	IS_iErrorSource = 0
	IS_iExternWarns_RF = 0
	IS_strErrorSource[] = "VW-User"
	RETURN TRUE
ENDIF
bOk = TRUE
;
; 1: Manuelle Messunganmeldung wurde verwendet
IF (iExternWarns B_AND IS_STATE_WARN_MANMEAS) == IS_STATE_WARN_MANMEAS THEN
	;bisher gibt es kein Flag
	bOk = FALSE
ENDIF
;
; 2: bei Ergebnissimulation
IF (iExternWarns B_AND IS_STATE_WARN_EVAL) == IS_STATE_WARN_EVAL THEN
	;bisher gibt es kein Flag
	bOk = FALSE
ENDIF
;
; 3: Toleranzverletzung
IF (iExternWarns B_AND IS_STATE_WARN_TOL) == IS_STATE_WARN_TOL THEN
	$FLAG[IS_FLAG_WARN_TOL] = TRUE
	bOk = FALSE
ENDIF
;
RETURN bOK
;
ENDFCT
;---------------------------------------------------------------------------------------------
;ENDFOLD
;
;FOLD Zentrale Funktion zur Fehlerbehandlung
;---------------------------------------------------------------------------------------------
DEF IS_ProcessErrors()
DECL CHAR strErrorSource[10]
DECL INT OFFSET
DECL STATE_T STATE
CHAR ch_tempString[300]
;
IF (IS_iExternErrors==0) AND (IS_iInternErrors==0) THEN
	RETURN
ENDIF
;
IF (IS_iExternErrors <> 0) THEN
	SWITCH IS_iErrorSource
	CASE 1
		strErrorSource[] = "RoVis"
		strErrorSource[6] = 0
	CASE 2
		strErrorSource[] = "Genesis"
		strErrorSource[8] = 0
	CASE 3
		strErrorSource[] = "IQRob"
		strErrorSource[6] = 0
	CASE 4
		strErrorSource[] = "ISRob"
		strErrorSource[6] = 0
	CASE 5
		strErrorSource[] = "Dynalog"
		strErrorSource[8] = 0
		SWITCH IS_iExternErrors
			CASE 1
				IS_MSG_ERR(IS_MSG_ERR_RTC_CALIB)
			CASE 2
				SWITCH IS_iServiceMode
				CASE IS_iTOOL_CHANGE
					IS_MSG_ERR(IS_MSG_ERR_RTC_CALC_TOOL)
				CASE IS_iROBOT_CHANGE
					IS_MSG_ERR(IS_MSG_ERR_RTC_CALC_BASE)
				CASE IS_iSENSOR_CHANGE_IMT
					IS_MSG_ERR(IS_MSG_ERR_SERV_SENSIMT)
				DEFAULT
					IS_MSG_ERR(IS_MSG_ERR_RTC)
				ENDSWITCH
			DEFAULT
				IS_MSG_ERR(IS_MSG_ERR_RTC)
			ENDSWITCH
		RETURN
	DEFAULT
		strErrorSource[] = "ISRA"
		strErrorSource[5] = 0
	ENDSWITCH
;
	OFFSET=0
	SWRITE(IS_strErrorSource[], STATE, OFFSET, "%s%d", strErrorSource[], IS_iExternErrors)
ENDIF
;
IF (IS_iInternErrors <> 0) THEN
	strErrorSource[] = "VW-User"
	strErrorSource[8]= 0
	OFFSET=0
	SWRITE(IS_strErrorSource[], STATE, OFFSET, "%s%d", strErrorSource[], IS_iInternErrors)
ENDIF
;
IF (IS_iInternErrors == IS_Err_ID_Tolerance) THEN
	OFFSET=0
	SWRITE(ch_tempString[], STATE, OFFSET, "Max = {X %.2f, Y %.2f, Z %.2f, A %.2f, B %.2f, C %.2f}", IS_CORR_ACCEPT_FRAME.X, IS_CORR_ACCEPT_FRAME.Y, IS_CORR_ACCEPT_FRAME.Z, IS_CORR_ACCEPT_FRAME.A, IS_CORR_ACCEPT_FRAME.B, IS_CORR_ACCEPT_FRAME.C)
	IS_MSG_ERR(IS_MSG_ERR_TOL_EXCEEDED)
	RETURN
ENDIF
;
SWITCH IS_iServiceMode
	CASE IS_iSENSOR_CHANGE
		IF (IS_iErrorSource==3) AND (IS_iExternErrors==16) THEN
			;IS_MSG_ERR(IS_MSG_ERR_SERV_SENS2)
			IS_MSG(IS_MSG_I_TRANS_AXES, IS_MSG_TYPE_NOTIFY) ;Achswinkel werden uebertragen
			IS_iFnctID = 0
		ELSE
		  ;IS_MSG_ERR(IS_MSG_ERR_SERV_SENS2)
		ENDIF
		RETURN
	CASE IS_iTOOL_CHANGE
		IF (IS_iErrorSource==3) AND (IS_iExternErrors==16) THEN
			;IS_MSG_ERR(IS_MSG_ERR_AXIS1A)
			IS_MSG(IS_MSG_I_TRANS_AXES, IS_MSG_TYPE_NOTIFY) ;Achswinkel werden uebertragen
			IS_iFnctID = 0
		ELSE
		  IS_MSG_ERR(IS_MSG_ERR_SERV_TOOL)
		ENDIF
		RETURN
	CASE IS_iROBOT_CHANGE
		IF (IS_iErrorSource==3) AND (IS_iExternErrors==16) THEN
			;IS_MSG_ERR(IS_MSG_ERR_AXIS1A)
			IS_MSG(IS_MSG_I_TRANS_AXES, IS_MSG_TYPE_NOTIFY) ;Achswinkel werden uebertragen
			IS_iFnctID = 0
		ELSE
		  IF (IS_iErrorSource==3) AND (IS_iExternErrors==32) THEN
		  	;IS_MSG_ERR(IS_MSG_ERR_AXIS1B)
				IS_MSG(IS_MSG_I_TRANS_BASE, IS_MSG_TYPE_NOTIFY) ;Basedaten werden uebertragen
				IS_iFnctID = 0
			ELSE
			  IF (IS_iErrorSource==3) AND (IS_iExternErrors==48) THEN
					;IS_MSG_ERR(IS_MSG_ERR_AXIS1B)
					;IS_MSG_ERR(IS_MSG_ERR_AXIS1A)
					IS_MSG(IS_MSG_I_TRANS_BASE, IS_MSG_TYPE_NOTIFY) ;Basedaten werden uebertragen)
					IS_MSG(IS_MSG_I_TRANS_AXES, IS_MSG_TYPE_NOTIFY) ;Achswinkel werden uebertragen
					IS_iFnctID = 0
			  ELSE
				  IS_MSG_ERR(IS_MSG_ERR_SERV_ROB)
				ENDIF
			ENDIF
		ENDIF
		RETURN
   CASE IS_iSENSOR_CHANGE_IMT
		IS_MSG_ERR(IS_MSG_ERR_SERV_SENSIMT)
		IS_iFnctID = 0
		RETURN
ENDSWITCH
;
SWITCH IS_iFnctID
;
;FOLD SNYC
CASE IS_FnctID_IMT_Sync1
	IF (IS_iExternErrors>0) THEN
		IS_MSG_ERR(IS_MSG_ERR_SYNC1A)
	ELSE
		IS_MSG_ERR(IS_MSG_ERR_SYNC1B)
	ENDIF
CASE IS_FnctID_IMT_Sync2
	IF (IS_iExternErrors>0) THEN
		IS_MSG_ERR(IS_MSG_ERR_SYNC2A)
	ELSE
		IS_MSG_ERR(IS_MSG_ERR_SYNC2B)
	ENDIF
;ENDFOLD (SYNC)
;
;FOLD SELECT
CASE IS_FnctID_IMT_SelectUp1
IF (IS_iExternErrors>0) THEN
	IF (IS_iErrorSource==3) AND ((IS_iExternErrors b_and 4)==4) THEN
		IS_MSG_ERR(IS_MSG_ERR_SELECT1A, IS_MODEL)
	ELSE
		IS_MSG_ERR(IS_MSG_ERR_SELECT1, IS_MODEL)
	ENDIF
ELSE
	SWITCH IS_iInternErrors
		CASE IS_Err_ID_Drain 																;Ablauffehler
			IS_MSG_ERR(IS_MSG_ERR_SELECT1B, IS_MODEL)
		CASE IS_Err_ID_Timeout 															;Timeout
			IS_MSG_ERR(IS_MSG_ERR_SELECT1C)
		DEFAULT
			IS_MSG_ERR(IS_MSG_ERR_SELECT1, IS_MODEL)
	ENDSWITCH
ENDIF
CASE IS_FnctID_IMT_SelectUp2
		SWITCH IS_iInternErrors
			CASE IS_Err_ID_Drain
				IS_MSG_ERR(IS_MSG_ERR_SELECT2A)
			CASE IS_Err_ID_ProgID
				IS_MSG_ERR(IS_MSG_ERR_SELECT2B, IS_PROGID)
			DEFAULT
				IS_MSG_ERR(IS_MSG_ERR_SELECT2)
		ENDSWITCH
CASE IS_FnctID_IMT_SelectUp3
		SWITCH IS_iInternErrors
			CASE IS_Err_ID_Timeout
				IS_MSG_ERR(IS_MSG_ERR_SELECT3A, IS_PROGID)
			DEFAULT
			 IS_MSG_ERR(IS_MSG_ERR_SELECT3, IS_PROGID)
		ENDSWITCH
;ENDFOLD (SELECT)
;
;FOLD IMT_RREPARE
CASE IS_FnctID_IMT_Prepare
	IF (IS_iExternErrors>0) THEN
		IF ((IS_iExternErrors b_and 8)==8) THEN
			IS_MSG_ERR(IS_MSG_ERR_IMT_PREPARE1A, IS_SUBTYP)
		ELSE
			IS_MSG_ERR(IS_MSG_ERR_IMT_PREPARE1, IS_SUBTYP)
		ENDIF
	ELSE
		SWITCH IS_iInternErrors
			CASE IS_Err_ID_Timeout
				IS_MSG_ERR(IS_MSG_ERR_IMT_PREPARE1B, IS_SUBTYP)
			DEFAULT
				IS_MSG_ERR(IS_MSG_ERR_IMT_PREPARE1, IS_SUBTYP)
		ENDSWITCH
	ENDIF
;ENDFOLD (IMT_RREPARE)
;
;FOLD IMT_APPLY
CASE IS_FnctID_IMT_Apply
	IS_MSG_ERR(IS_MSG_ERR_IMT_APPLY, IS_SUBTYP)
;ENDFOLD (IMT_APPLY)
;
;FOLD ACHSWINKEL SENDEN
CASE IS_FnctID_IMT_SendAxis1
	IF (IS_iExternErrors>0) THEN
		IF ((IS_iExternErrors b_and 8)==8) THEN
			IS_MSG_ERR(IS_MSG_ERR_IMT_PREPARE1, IS_SUBTYP)
			IS_iFnctID = 0
			RETURN
		ENDIF
		IF (IS_iErrorSource==3) AND (IS_iExternErrors==16) THEN
		  IF (($MODE_OP==#T2) OR ($MODE_OP==#T1)) THEN
        ;MsgNotify("Achswinkel werden uebertragen", "ISRA")
      ENDIF
		ELSE
		  IF (IS_iErrorSource==3) AND (IS_iExternErrors==32) THEN
        IF (($MODE_OP==#T2) OR ($MODE_OP==#T1)) THEN
           ;MsgNotify("Basedaten werden uebertragen", "ISRA")
        ENDIF
			ELSE
			 IF (IS_iErrorSource==3) AND (IS_iExternErrors==48) THEN
         IF (($MODE_OP==#T2) OR ($MODE_OP==#T1)) THEN
            ;MsgNotify("Basedaten und Achswinkel werden uebertragen", "ISRA")
         ENDIF
			 ELSE
					IS_MSG_ERR(IS_MSG_ERR_AXIS1)
				ENDIF
			ENDIF
		ENDIF
	ELSE
		SWITCH IS_iInternErrors
			CASE IS_Err_ID_Drain
				IS_MSG_ERR(IS_MSG_ERR_AXIS1C)
			CASE IS_Err_ID_Timeout
				IS_MSG_ERR(IS_MSG_ERR_AXIS1D)
			DEFAULT
				IS_MSG_ERR(IS_MSG_ERR_AXIS1)
		ENDSWITCH
	ENDIF
CASE IS_FnctID_IMT_SendAxis2
	IF (IS_iExternErrors>0) THEN
		IF (IS_iErrorSource==3) AND (IS_iExternErrors==32) THEN
			IS_MSG_ERR(IS_MSG_ERR_AXIS1B)
		ELSE
			IS_MSG_ERR(IS_MSG_ERR_AXIS2)
		ENDIF
	ELSE
		SWITCH IS_iInternErrors
			CASE IS_Err_ID_Drain
				IS_MSG_ERR(IS_MSG_ERR_AXIS2A)
			CASE IS_Err_ID_Timeout
				IS_MSG_ERR(IS_MSG_ERR_AXIS2B)
			DEFAULT
				IS_MSG_ERR(IS_MSG_ERR_AXIS2)
		ENDSWITCH
	ENDIF
CASE IS_FnctID_IMT_SendAxis3
	IF (IS_iExternErrors>0) THEN
		IS_MSG_ERR(IS_MSG_ERR_AXIS3)
	ELSE
		SWITCH IS_iInternErrors
			CASE IS_Err_ID_Drain
				IS_MSG_ERR(IS_MSG_ERR_AXIS3A)
			CASE IS_Err_ID_Timeout
				IS_MSG_ERR(IS_MSG_ERR_AXIS3B)
			DEFAULT
				IS_MSG_ERR(IS_MSG_ERR_AXIS3)
		ENDSWITCH
	ENDIF
CASE IS_FnctID_IMT_SendAxis4
	IF (IS_iExternErrors>0) THEN
		IS_MSG_ERR(IS_MSG_ERR_AXIS4)
	ELSE
		SWITCH IS_iInternErrors
			CASE IS_Err_ID_Drain
				IS_MSG_ERR(IS_MSG_ERR_AXIS4A)
			CASE IS_Err_ID_Timeout
				IS_MSG_ERR(IS_MSG_ERR_AXIS4B)
			DEFAULT
				IS_MSG_ERR(IS_MSG_ERR_AXIS4)
		ENDSWITCH
	ENDIF
;ENDFOLD (ACHSEN)
;
;FOLD BASE SENDEN
CASE IS_FnctID_IMT_SendBase1
	IF (IS_iExternErrors>0) THEN
		IS_MSG_ERR(IS_MSG_ERR_BASE1)
	ELSE
		SWITCH IS_iInternErrors
			CASE IS_Err_ID_Drain
				IS_MSG_ERR(IS_MSG_ERR_BASE1A)
			CASE IS_Err_ID_Timeout
				IS_MSG_ERR(IS_MSG_ERR_BASE2B)
			DEFAULT
				IS_MSG_ERR(IS_MSG_ERR_BASE1)
		ENDSWITCH
	ENDIF
CASE IS_FnctID_IMT_SendBase2
	IF (IS_iExternErrors>0) THEN
		IS_MSG_ERR(IS_MSG_ERR_BASE2)
	ELSE
		SWITCH IS_iInternErrors
			CASE IS_Err_ID_Drain
				IS_MSG_ERR(IS_MSG_ERR_BASE2A)
			CASE IS_Err_ID_Timeout
				IS_MSG_ERR(IS_MSG_ERR_BASE2B)
			DEFAULT
				IS_MSG_ERR(IS_MSG_ERR_BASE2)
		ENDSWITCH
	ENDIF
CASE IS_FnctID_IMT_SendBase3
	IF (IS_iExternErrors>0) THEN
		IS_MSG_ERR(IS_MSG_ERR_BASE3)
	ELSE
		SWITCH IS_iInternErrors
			CASE IS_Err_ID_Drain
				IS_MSG_ERR(IS_MSG_ERR_BASE3A)
			CASE IS_Err_ID_Timeout
				IS_MSG_ERR(IS_MSG_ERR_BASE3B)
			DEFAULT
				IS_MSG_ERR(IS_MSG_ERR_BASE3)
		ENDSWITCH
	ENDIF
;ENDFOLD (BASE SENDEN)
;
;FOLD POSE SENDEN
CASE IS_FnctID_IMT_SendPose1
	IF (IS_iExternErrors>0) THEN
		IS_MSG_ERR(IS_MSG_ERR_POSE1)
	ELSE
		SWITCH IS_iInternErrors
			CASE IS_Err_ID_Drain
				IS_MSG_ERR(IS_MSG_ERR_POSE1A)
			CASE IS_Err_ID_Timeout
				IS_MSG_ERR(IS_MSG_ERR_POSE1B)
			DEFAULT
				IS_MSG_ERR(IS_MSG_ERR_POSE1)
		ENDSWITCH
	ENDIF
CASE IS_FnctID_IMT_SendPose2
	IF (IS_iExternErrors>0) THEN
		IS_MSG_ERR(IS_MSG_ERR_POSE2)
	ELSE
		SWITCH IS_iInternErrors
			CASE IS_Err_ID_Drain
				IS_MSG_ERR(IS_MSG_ERR_POSE2A)
			CASE IS_Err_ID_Timeout
				IS_MSG_ERR(IS_MSG_ERR_POSE2B)
			DEFAULT
				IS_MSG_ERR(IS_MSG_ERR_POSE2)
		ENDSWITCH
	ENDIF
CASE IS_FnctID_IMT_SendPose3
	IF (IS_iExternErrors>0) THEN
		IS_MSG_ERR(IS_MSG_ERR_POSE3)
	ELSE
		SWITCH IS_iInternErrors
			CASE IS_Err_ID_Drain
				IS_MSG_ERR(IS_MSG_ERR_POSE3A)
			CASE IS_Err_ID_Timeout
				IS_MSG_ERR(IS_MSG_ERR_POSE3B)
			DEFAULT
				IS_MSG_ERR(IS_MSG_ERR_POSE3)
		ENDSWITCH
	ENDIF
;ENDFOLD (POSE SENDEN)
;
;FOLD TOOL SENDEN
CASE IS_FnctID_IMT_SendTool1
	IF (IS_iExternErrors>0) THEN
		IS_MSG_ERR(IS_MSG_ERR_TOOL1)
	ELSE
		SWITCH IS_iInternErrors
			CASE IS_Err_ID_Drain
				IS_MSG_ERR(IS_MSG_ERR_TOOL1A)
			CASE IS_Err_ID_Timeout
				IS_MSG_ERR(IS_MSG_ERR_TOOL1B)
			DEFAULT
				IS_MSG_ERR(IS_MSG_ERR_TOOL1)
		ENDSWITCH
	ENDIF
CASE IS_FnctID_IMT_SendTool2
	IF (IS_iExternErrors>0) THEN
		IS_MSG_ERR(IS_MSG_ERR_TOOL2)
	ELSE
		SWITCH IS_iInternErrors
			CASE IS_Err_ID_Drain
				IS_MSG_ERR(IS_MSG_ERR_TOOL2A)
			CASE IS_Err_ID_Timeout
				IS_MSG_ERR(IS_MSG_ERR_TOOL2B)
			DEFAULT
				IS_MSG_ERR(IS_MSG_ERR_TOOL2)
		ENDSWITCH
	ENDIF
CASE IS_FnctID_IMT_SendTool3
	IF (IS_iExternErrors>0) THEN
		IS_MSG_ERR(IS_MSG_ERR_TOOL3)
	ELSE
		SWITCH IS_iInternErrors
			CASE IS_Err_ID_Drain
				IS_MSG_ERR(IS_MSG_ERR_TOOL3A)
			CASE IS_Err_ID_Timeout
				IS_MSG_ERR(IS_MSG_ERR_TOOL3B)
			DEFAULT
				IS_MSG_ERR(IS_MSG_ERR_TOOL3)
		ENDSWITCH
	ENDIF
;ENDFOLD (POSE SENDEN)
;
;FOLD END_POSE
CASE IS_FnctID_IMT_EndPose1, IS_FnctID_IMT_EndPose2
	IF (IS_iExternErrors>0) THEN
		IF ((IS_iExternErrors B_AND 64)==64) THEN
			IS_MSG_ERR(IS_MSG_ERR_IMT_END1A)
		ENDIF
		IF ((IS_iExternErrors B_AND 128)==128) THEN
			IS_MSG_ERR(IS_MSG_ERR_IMT_END1B)
		ELSE
			IS_MSG_ERR(IS_MSG_ERR_IMT_END1)
		ENDIF
	ELSE
		SWITCH IS_iInternErrors
			CASE IS_Err_ID_Timeout
				IS_MSG_ERR(IS_MSG_ERR_IMT_END1C)
			DEFAULT
				IS_MSG_ERR(IS_MSG_ERR_IMT_END1)
		ENDSWITCH
	ENDIF
;ENDFOLD (END_POSE)
;
;FOLD GetCorr
CASE IS_FnctID_IMT_GetCorr1
	IF (IS_iExternErrors>0) THEN
			IS_MSG_ERR(IS_MSG_ERR_GETCORR1)
	ELSE
		SWITCH IS_iInternErrors
			CASE IS_Err_ID_Drain
				IS_MSG_ERR(IS_MSG_ERR_GETCORR1A)
			CASE IS_Err_ID_Timeout
				IS_MSG_ERR(IS_MSG_ERR_GETCORR1B)
			DEFAULT
				IS_MSG_ERR(IS_MSG_ERR_GETCORR1)
		ENDSWITCH
	ENDIF
CASE IS_FnctID_IMT_GetCorr2
	IF (IS_iExternErrors>0) THEN
			IS_MSG_ERR(IS_MSG_ERR_GETCORR2)
	ELSE
		SWITCH IS_iInternErrors
			CASE IS_Err_ID_Drain
				IS_MSG_ERR(IS_MSG_ERR_GETCORR2A)
			CASE IS_Err_ID_Timeout
				IS_MSG_ERR(IS_MSG_ERR_GETCORR2B)
			DEFAULT
				IS_MSG_ERR(IS_MSG_ERR_GETCORR2)
		ENDSWITCH
	ENDIF
CASE IS_FnctID_IMT_GetCorr3
	IF (IS_iExternErrors>0) THEN
			IS_MSG_ERR(IS_MSG_ERR_GETCORR3)
	ELSE
		SWITCH IS_iInternErrors
			CASE IS_Err_ID_Drain
				IS_MSG_ERR(IS_MSG_ERR_GETCORR3A)
			CASE IS_Err_ID_Timeout
				IS_MSG_ERR(IS_MSG_ERR_GETCORR3B)
			DEFAULT
				IS_MSG_ERR(IS_MSG_ERR_GETCORR3)
		ENDSWITCH
	ENDIF
CASE IS_FnctID_IMT_GetCorr4
	IF (IS_iInternErrors == IS_Err_ID_Timeout) THEN
		IS_MSG_ERR(IS_MSG_ERR_GETCORR4A)
	ELSE
		IS_MSG_ERR(IS_MSG_ERR_GETCORR4)
	ENDIF
;ENDFOLD (GetCorr)
;
;FOLD RF_INIT
CASE IS_FnctID_RF_Init1
	IS_MSG_ERR(IS_MSG_ERR_RF_INIT1A)
CASE IS_FnctID_RF_Init2
	IS_MSG_ERR(IS_MSG_ERR_RF_INIT2A)
;ENDFOLD (RF_INIT)
;
;FOLD RF_Prepare
CASE IS_FnctID_RF_Prepare1
	IF (IS_iExternErrors>0) THEN
		IS_MSG_ERR(IS_MSG_ERR_RF_PREPARE1A, IS_TYP, IS_SUBTYP)
	ELSE
		IF (IS_iInternErrors == IS_Err_ID_Timeout) THEN
			IS_MSG_ERR(IS_MSG_ERR_RF_PREPARE1B, IS_TYP, IS_SUBTYP)
		ELSE
			IS_MSG_ERR(IS_MSG_ERR_RF_PREPARE1, IS_TYP, IS_SUBTYP)
		ENDIF
	ENDIF
CASE IS_FnctID_RF_Prepare2
	IF (IS_iExternErrors>0) THEN
		IS_MSG_ERR(IS_MSG_ERR_RF_PREPARE2A, IS_TYP, IS_SUBTYP)
	ELSE
		IF (IS_iInternErrors == IS_Err_ID_Timeout) THEN
			IS_MSG_ERR(IS_MSG_ERR_RF_PREPARE2B, IS_TYP, IS_SUBTYP)
		ELSE
			IS_MSG_ERR(IS_MSG_ERR_RF_PREPARE2, IS_TYP, IS_SUBTYP)
		ENDIF
	ENDIF
CASE IS_FnctID_RF_Prepare3
	IF (IS_iExternErrors>0) THEN
		IF ((IS_iExternErrors b_and IS_ErrBit_Prepare)==IS_ErrBit_Prepare) THEN
			IS_MSG_ERR(IS_MSG_ERR_RF_PREPARE3A, IS_TYP, IS_SUBTYP)
		ELSE
			IS_MSG_ERR(IS_MSG_ERR_RF_PREPARE3B, IS_TYP, IS_SUBTYP)
		ENDIF
	ELSE
		IF (IS_iInternErrors == IS_Err_ID_Timeout) THEN
			IS_MSG_ERR(IS_MSG_ERR_RF_PREPARE3C, IS_TYP, IS_SUBTYP)
		ELSE
			IS_MSG_ERR(IS_MSG_ERR_RF_PREPARE3, IS_TYP, IS_SUBTYP)
		ENDIF
	ENDIF
;ENDFOLD (RF_Prepare)
;
;FOLD RF_APPLY
CASE IS_FnctID_RF_Apply1
	IS_MSG_ERR(IS_MSG_ERR_RF_APPLY1, IS_TYP, IS_SUBTYP)
CASE IS_FnctID_RF_Apply2
	IF (IS_iExternErrors>0) THEN
			IS_MSG_ERR(IS_MSG_ERR_RF_APPLY2B, IS_TYP, IS_SUBTYP)
	ELSE
		IF (IS_iInternErrors == IS_Err_ID_Timeout) THEN
			IS_MSG_ERR(IS_MSG_ERR_RF_APPLY2A, IS_TYP, IS_SUBTYP)
		ELSE
			IS_MSG_ERR(IS_MSG_ERR_RF_APPLY2, IS_TYP, IS_SUBTYP)
		ENDIF
	ENDIF
CASE IS_FnctID_RF_Apply3
	IF (IS_iExternErrors>0) THEN
		IF ((IS_iExternErrors b_and IS_ErrBit_Feature)==IS_ErrBit_Feature) THEN
			IS_MSG_ERR(IS_MSG_ERR_RF_APPLY3C, IS_TYP, IS_SUBTYP)
			;IS_iFnctID = 0
			;RETURN
		ELSE
			IF ((IS_iExternErrors b_and IS_ErrBit_Tol)==IS_ErrBit_Tol) THEN
				IS_MSG_ERR(IS_MSG_ERR_RF_APPLY3D, IS_TYP, IS_SUBTYP)
				;IS_iFnctID = 0
				;RETURN
			ELSE
				IF ((IS_iExternErrors b_and IS_ErrBit_Deadly)==IS_ErrBit_Deadly) THEN
					IS_MSG_ERR(IS_MSG_ERR_RF_APPLY3E, IS_TYP, IS_SUBTYP)
					;IS_iFnctID = 0
					;RETURN
				ELSE
					IS_MSG_ERR(IS_MSG_ERR_RF_APPLY3B, IS_TYP, IS_SUBTYP)
				ENDIF
			ENDIF
		ENDIF
	ELSE
		IF (IS_iInternErrors == IS_Err_ID_Timeout) THEN
			IS_MSG_ERR(IS_MSG_ERR_RF_APPLY3A, IS_TYP, IS_SUBTYP)
		ELSE
			IS_MSG_ERR(IS_MSG_ERR_RF_APPLY3, IS_TYP, IS_SUBTYP)
		ENDIF
	ENDIF
CASE IS_FnctID_RF_Apply4
	IF (IS_iExternErrors>0) THEN
		IF ((IS_iExternErrors b_and IS_ErrBit_Feature)==IS_ErrBit_Feature) THEN
			IS_MSG_ERR(IS_MSG_ERR_RF_APPLY4C, IS_TYP, IS_SUBTYP)
			;IS_iFnctID = 0
			;RETURN
		ELSE
			IF ((IS_iExternErrors b_and IS_ErrBit_Tol)==IS_ErrBit_Tol) THEN
				IS_MSG_ERR(IS_MSG_ERR_RF_APPLY4D, IS_TYP, IS_SUBTYP)
				;IS_iFnctID = 0
				;RETURN
			ELSE
				IF ((IS_iExternErrors b_and IS_ErrBit_Deadly)==IS_ErrBit_Deadly) THEN
					IS_MSG_ERR(IS_MSG_ERR_RF_APPLY4E, IS_TYP, IS_SUBTYP)
					;IS_iFnctID = 0
					;RETURN
				ELSE
					IS_MSG_ERR(IS_MSG_ERR_RF_APPLY4B, IS_TYP, IS_SUBTYP)
				ENDIF
			ENDIF
		ENDIF
	ELSE
		IF (IS_iInternErrors == IS_Err_ID_Timeout) THEN
			IS_MSG_ERR(IS_MSG_ERR_RF_APPLY4A, IS_TYP, IS_SUBTYP)
		ELSE
			IS_MSG_ERR(IS_MSG_ERR_RF_APPLY4, IS_TYP, IS_SUBTYP)
		ENDIF
	ENDIF
CASE IS_FnctID_RF_Apply5
	IF (IS_iExternErrors>0) THEN
		IF ((IS_iExternErrors b_and IS_ErrBit_Feature)==IS_ErrBit_Feature) THEN
			IS_MSG_ERR(IS_MSG_ERR_RF_APPLY5C, IS_TYP, IS_SUBTYP)
			;IS_iFnctID = 0
			;RETURN
		ELSE
			IF ((IS_iExternErrors b_and IS_ErrBit_Tol)==IS_ErrBit_Tol) THEN
				IS_MSG_ERR(IS_MSG_ERR_RF_APPLY5D, IS_TYP, IS_SUBTYP)
				;IS_iFnctID = 0
				;RETURN
			ELSE
				IF ((IS_iExternErrors b_and IS_ErrBit_Deadly)==IS_ErrBit_Deadly) THEN
					IS_MSG_ERR(IS_MSG_ERR_RF_APPLY5E, IS_TYP, IS_SUBTYP)
					;IS_iFnctID = 0
					;RETURN
				ELSE
					IS_MSG_ERR(IS_MSG_ERR_RF_APPLY5B, IS_TYP, IS_SUBTYP)
				ENDIF
			ENDIF
		ENDIF
	ELSE
		IF (IS_iInternErrors == IS_Err_ID_Timeout) THEN
			IS_MSG_ERR(IS_MSG_ERR_RF_APPLY5A, IS_TYP, IS_SUBTYP)
		ELSE
			IS_MSG_ERR(IS_MSG_ERR_RF_APPLY5, IS_TYP, IS_SUBTYP)
		ENDIF
	ENDIF
CASE IS_FnctID_RF_Apply6
	IS_MSG_ERR(IS_MSG_ERR_RF_APPLY6)
;ENDFOLD (RF_APPLY)
;
;FOLD RF_ENDPOSE
CASE IS_FnctID_RF_End1
	IF (IS_iExternErrors>0) THEN
		IF ((IS_iExternErrors b_and IS_ErrBit_Feature)==IS_ErrBit_Feature) THEN
			IS_MSG_ERR(IS_MSG_ERR_RF_END1B)
			;IS_iFnctID = 0
			;RETURN
		ELSE
			IF ((IS_iExternErrors b_and IS_ErrBit_Tol)==IS_ErrBit_Tol) THEN
				IS_MSG_ERR(IS_MSG_ERR_RF_END1C)
				;IS_iFnctID = 0
				;RETURN
			ELSE
				IF ((IS_iExternErrors b_and IS_ErrBit_Deadly)==IS_ErrBit_Deadly) THEN
					IS_MSG_ERR(IS_MSG_ERR_RF_END1E)
					;IS_iFnctID = 0
					;RETURN
				ELSE
					IS_MSG_ERR(IS_MSG_ERR_RF_END1A)
				ENDIF
			ENDIF
		ENDIF
	ELSE
		IF (IS_iInternErrors == IS_Err_ID_Timeout) THEN
			IS_MSG_ERR(IS_MSG_ERR_RF_END1D)
		ELSE
			IS_MSG_ERR(IS_MSG_ERR_RF_END1)
		ENDIF
	ENDIF
CASE IS_FnctID_RF_End2
	IF (IS_iExternErrors>0) THEN
		IF ((IS_iExternErrors b_and IS_ErrBit_Feature)==IS_ErrBit_Feature) THEN
			IS_MSG_ERR(IS_MSG_ERR_RF_END2B)
			;IS_iFnctID = 0
			;RETURN
		ELSE
			IF ((IS_iExternErrors b_and IS_ErrBit_Tol)==IS_ErrBit_Tol) THEN
				IS_MSG_ERR(IS_MSG_ERR_RF_END2C)
				;IS_iFnctID = 0
				;RETURN
			ELSE
				IF ((IS_iExternErrors b_and IS_ErrBit_Deadly)==IS_ErrBit_Deadly) THEN
					IS_MSG_ERR(IS_MSG_ERR_RF_END2E)
					;IS_iFnctID = 0
					;RETURN
				ELSE
					IS_MSG_ERR(IS_MSG_ERR_RF_END2A)
				ENDIF
			ENDIF
		ENDIF
	ELSE
		IF (IS_iInternErrors == IS_Err_ID_Timeout) THEN
			IS_MSG_ERR(IS_MSG_ERR_RF_END2D)
		ELSE
			IS_MSG_ERR(IS_MSG_ERR_RF_END2)
		ENDIF
	ENDIF
CASE IS_FnctID_RF_End2
	IS_MSG_ERR(IS_MSG_ERR_RF_END3)
;ENDFOLD (RF_ENDPOSE)
;
;FOLD RF_GETGORR
CASE IS_FnctID_RF_GCorr1
	IF (IS_iExternErrors>0) THEN
		IS_MSG_ERR(IS_MSG_ERR_RF_CORR1B)
	ELSE
		IF (IS_iInternErrors == IS_Err_ID_Timeout) THEN
			IS_MSG_ERR(IS_MSG_ERR_RF_CORR1A)
		ELSE
			IS_MSG_ERR(IS_MSG_ERR_RF_END1)
		ENDIF
	ENDIF
CASE IS_FnctID_RF_GCorr2
	IF (IS_iExternErrors>0) THEN
		IS_MSG_ERR(IS_MSG_ERR_RF_CORR2B)
	ELSE
		IF (IS_iInternErrors == IS_Err_ID_Timeout) THEN
			IS_MSG_ERR(IS_MSG_ERR_RF_CORR2A)
		ELSE
			IS_MSG_ERR(IS_MSG_ERR_RF_END2)
		ENDIF
	ENDIF
CASE IS_FnctID_RF_GCorr3
	IS_MSG_ERR(IS_MSG_ERR_RF_CORR3)
;ENDFOLD (RF_GETGORR)
;
;FOLD Service
CASE IS_FnctID_IMT_Service
	IF (IS_iInternErrors == IS_Err_ID_Timeout) THEN
		SWITCH IS_iServiceMode
			CASE IS_iSENSOR_CHANGE
				IS_MSG_ERR(IS_MSG_ERR_SERVICE1a)
			CASE IS_iTOOL_CHANGE
				IS_MSG_ERR(IS_MSG_ERR_SERVICE1b)
			CASE IS_iROBOT_CHANGE
				IS_MSG_ERR(IS_MSG_ERR_SERVICE1c)
			CASE IS_iSENSOR_CHANGE_IMT
				IS_MSG_ERR(IS_MSG_ERR_SERVICE1d)
		ENDSWITCH
	ELSE
		SWITCH IS_iServiceMode
			CASE IS_iSENSOR_CHANGE
				IS_MSG_ERR(IS_MSG_ERR_SERVICE1e)
			CASE IS_iTOOL_CHANGE
				IS_MSG_ERR(IS_MSG_ERR_SERVICE1f)
			CASE IS_iROBOT_CHANGE
				IS_MSG_ERR(IS_MSG_ERR_SERVICE1g)
			CASE IS_iSENSOR_CHANGE_IMT
				IS_MSG_ERR(IS_MSG_ERR_SERVICE1h)
		ENDSWITCH
	ENDIF
;ENDFOLD (Service)
;
;FOLD ProcessState
CASE IS_FnctID_IMT_GetExtStat
	IS_MSG_ERR(IS_MSG_ERR_IMT_APPLY, IS_SUBTYP)
;ENDFOLD (ProcessState)
;
ENDSWITCH
;
IS_iFnctID = 0
;
END
;---------------------------------------------------------------------------------------------
;ENDFOLD
;
;FOLD Ergebnis-Zustand abfragen
;---------------------------------------------------------------------------------------------
DEFFCT BOOL IS_IMT_GetExternState (iStateResult:OUT, iStateWarning:OUT)
DECL INT iStateResult
DECL INT iStateWarning
DECL BOOL b_RetVal
;
IS_iFnctID = IS_FnctID_IMT_GetExtStat
;
IS_TX8_DATA_ID 				= 58			;Zustandsabfrage
IS_TX1_DATA_REQUEST 	= TRUE
IS_TX1_HANDSHAKE 			= IS_ToggleHandshake()
;
IF (IS_Wait(#IS_ERROR_ID, TRUE, 0) == FALSE) THEN
	$FLAG[IS_FLAG_ERROR] = TRUE
	IS_SetInternError(IS_IntErr_StReq1)
	RETURN FALSE
ENDIF
;
IS_iErrorSource  	= IS_RX8_ERR_SYS_ID
IS_iExternErrors 	= IS_RX8_ERRORS
iStateResult  		= IS_RX8_STATE_RESULT
iStateWarning 		= IS_RX8_STATE_WARNING
;
IS_TX1_DATA_REQUEST 	= FALSE
IS_TX1_DATA_ACCEPTED 	= TRUE
IS_TX1_HANDSHAKE 			= IS_ToggleHandshake()
;
b_RetVal = IS_Wait(#IS_ERROR_ID, FALSE, 0)
;
IF (b_RetVal == FALSE) THEN
	$FLAG[IS_FLAG_ERROR] = TRUE
	IS_SetInternError(IS_IntErr_StReq2)
ENDIF
;
IS_TX8_DATA_ID 				= 0
IS_TX1_DATA_ACCEPTED 	= FALSE
;
RETURN b_RetVal
ENDFCT
;---------------------------------------------------------------------------------------------
;ENDFOLD
;
;FOLD Ergebniszustand auf Roboter Flags abbilden
;---------------------------------------------------------------------------------------------
DEFFCT BOOL IS_IMT_ProcessExtState (iExternStateResult:IN, iExternStateWarning:IN)
DECL INT iExternStateResult
DECL INT iExternStateWarning
;
IF (iExternStateResult B_AND IS_STATE_RESULT_OK) == IS_STATE_RESULT_OK THEN
	$FLAG[IS_FLAG_RESULT_OK]  = TRUE
	$FLAG[IS_FLAG_RESULT_NOK] = FALSE
ELSE
	$FLAG[IS_FLAG_RESULT_OK]	= FALSE
ENDIF
;
IF (iExternStateResult B_AND IS_STATE_RESULT_NOK) == IS_STATE_RESULT_NOK THEN
	$FLAG[IS_FLAG_RESULT_NOK] = TRUE
	$FLAG[IS_FLAG_RESULT_OK]  = FALSE
  IS_MSG_ERR(IS_MSG_RESULT_NOK)
  RETURN FALSE
ELSE
	$FLAG[IS_FLAG_RESULT_NOK]	= FALSE
  $FLAG[IS_FLAG_RESULT_OK]  = TRUE
ENDIF
;
IF (iExternStateWarning B_AND IS_STATE_WARN_TOL) == IS_STATE_WARN_TOL THEN
 	$FLAG[IS_FLAG_WARN_TOL] = TRUE
ELSE
  $FLAG[IS_FLAG_WARN_TOL] = FALSE
ENDIF
;
RETURN TRUE
ENDFCT
;---------------------------------------------------------------------------------------------
;ENDFOLD
;
;FOLD Systemdiagnose durchfuehren
;---------------------------------------------------------------------------------------------
DEF  IS_SYSTEM_DIAG ()
DECL BOOL bFlag
;
IF (IS_SYS_TYPE == IS_SYS_TYPE_IMT) THEN
	IF $IS_LIVE_SIGNAL THEN
		IS_MSG(IS_MSG_I_SYS_DIAG_1, IS_MSG_TYPE_NOTIFY)
	ELSE
		IS_MSG(IS_MSG_I_SYS_DIAG_2, IS_MSG_TYPE_NOTIFY)
		RETURN
	ENDIF
	;
	IF $IS_COMMUNICATE THEN
		IS_MSG(IS_MSG_I_SYS_DIAG_3, IS_MSG_TYPE_NOTIFY)
	ELSE
		IS_MSG(IS_MSG_I_SYS_DIAG_4, IS_MSG_TYPE_NOTIFY)
	ENDIF
	;
	;IS_MSG(0,7)
	IS_MSG(IS_MSG_I_SYNC, IS_MSG_TYPE_DIALOG)
	;
	IF (IS_ANSWER==1) THEN
		$IS_COMMUNICATE = TRUE
		IF IS_IMT_SyncHandshake() THEN
			IS_MSG(IS_MSG_I_SYS_DIAG_5, IS_MSG_TYPE_NOTIFY)
		ELSE
			IS_MSG(IS_MSG_I_SYS_DIAG_6, IS_MSG_TYPE_NOTIFY)
		ENDIF
	ELSE
		IS_MSG(IS_MSG_I_SYS_DIAG_7, IS_MSG_TYPE_NOTIFY)
	ENDIF
	;
ENDIF
;
IF (IS_SYS_TYPE == IS_SYS_TYPE_RF) THEN
	IF $IS_COMMUNICATE THEN
		IS_MSG(IS_MSG_I_SYS_DIAG_3, IS_MSG_TYPE_NOTIFY)
	ELSE
		IS_MSG(IS_MSG_I_SYS_DIAG_4, IS_MSG_TYPE_NOTIFY)
	ENDIF
	;
	;IS_MSG (0,7)
	IS_MSG(IS_MSG_I_SYNC, IS_MSG_TYPE_DIALOG)
	;
	IF (IS_ANSWER==1) THEN
		$IS_COMMUNICATE = TRUE
		;
		ISRA_PG_INIT()
		;
		IF IS_State_OK() THEN
			IS_MSG(IS_MSG_I_SYS_DIAG_5, IS_MSG_TYPE_NOTIFY)
		ELSE
			IS_MSG(IS_MSG_I_SYS_DIAG_6, IS_MSG_TYPE_NOTIFY)
		ENDIF
	ELSE
		IS_MSG(IS_MSG_I_SYS_DIAG_7, IS_MSG_TYPE_NOTIFY)
	ENDIF
ENDIF
;
END
;---------------------------------------------------------------------------------------------
;ENDFOLD
;
;
;FOLD HW über separate Messung prüfen
;---------------------------------------------------------------------------------------------
DEF IS_CheckHW()
	IF ((NOT IS_STATE_OK()) AND (NOT IS_bHWCheckMode) AND $IS_LIVE_SIGNAL) THEN
		;MsgNotify("IS_CheckHW", "Executing")
		; Fehlerflags speichern
		IS_SaveErrorFlags()
		;
		ISRA_PG_INIT()
		IS_bHWCheckMode = TRUE
		;
    IS_RF_Prepare(99, 0, 0)
    IS_RF_Apply(0)
    IS_RF_EndPose()
		;
		IF (NOT IS_STATE_OK()) AND (IS_RX1_RF_ERR_FEAT == TRUE) THEN
			$FLAG[IS_FLAG_ERR_ACQ] = TRUE
			$FLAG[IS_FLAG_ERROR] = TRUE
			IS_bHWCheckMode = FALSE
			IS_MSG_ERR(IS_MSG_ERR_RF_APPLY3E)
			;MsgNotify("IS_CheckHW","HW Error detected")
		ELSE
			IS_RestoreErrorFlags()
		ENDIF
	ENDIF
	IS_bHWCheckMode = FALSE
END
;---------------------------------------------------------------------------------------------
;ENDFOLD
;
;FOLD Speichern der Fehlerflags
;---------------------------------------------------------------------------------------------
DEF IS_SaveErrorFlags()
;
IS_FLAGS_SAVED[1] = $FLAG[IS_FLAG_ERR_SPS]
IS_FLAGS_SAVED[2] = $FLAG[IS_FLAG_ERR_ROBOT]
IS_FLAGS_SAVED[3] = $FLAG[IS_FLAG_ERR_PREPARE]
IS_FLAGS_SAVED[4] = $FLAG[IS_FLAG_ERR_ACQ]
IS_FLAGS_SAVED[5] = $FLAG[IS_FLAG_ERR_FEATURE]
IS_FLAGS_SAVED[6] = $FLAG[IS_FLAG_ERR_EVAL]
IS_FLAGS_SAVED[7] = $FLAG[IS_FLAG_ERR_TOL]
IS_FLAGS_SAVED[8] = $FLAG[IS_FLAG_WARN_TOL]
IS_FLAGS_SAVED[9] = $FLAG[IS_FLAG_KAL1_HLP]
IS_FLAGS_SAVED[10] = $FLAG[IS_FLAG_KAL2_HLP]
IS_FLAGS_SAVED[11] = $FLAG[IS_FLAG_RESULT_OK]
IS_FLAGS_SAVED[12] = $FLAG[IS_FLAG_RESULT_NOK]
IS_FLAGS_SAVED[13] = $FLAG[IS_FLAG_ERROR]
;
END
;---------------------------------------------------------------------------------------------
;ENDFOLD
;
;FOLD Wiederherstellen der Fehlerflags
;---------------------------------------------------------------------------------------------
DEF IS_RestoreErrorFlags()
;
$FLAG[IS_FLAG_ERR_SPS] 		= IS_FLAGS_SAVED[1]
$FLAG[IS_FLAG_ERR_ROBOT] 	= IS_FLAGS_SAVED[2]
$FLAG[IS_FLAG_ERR_PREPARE]= IS_FLAGS_SAVED[3]
$FLAG[IS_FLAG_ERR_ACQ]		= IS_FLAGS_SAVED[4]
$FLAG[IS_FLAG_ERR_FEATURE]= IS_FLAGS_SAVED[5]
$FLAG[IS_FLAG_ERR_EVAL]		= IS_FLAGS_SAVED[6]
$FLAG[IS_FLAG_ERR_TOL]		= IS_FLAGS_SAVED[7]
$FLAG[IS_FLAG_WARN_TOL]		= IS_FLAGS_SAVED[8]
$FLAG[IS_FLAG_KAL1_HLP]		= IS_FLAGS_SAVED[9]
$FLAG[IS_FLAG_KAL2_HLP]		= IS_FLAGS_SAVED[10]
$FLAG[IS_FLAG_RESULT_OK]	= IS_FLAGS_SAVED[11]
$FLAG[IS_FLAG_RESULT_NOK]	= IS_FLAGS_SAVED[12]
$FLAG[IS_FLAG_ERROR]			= IS_FLAGS_SAVED[13]
;
END
;---------------------------------------------------------------------------------------------
;ENDFOLD
;
;
;FOLD Fehlermeldungen deutsch
;---------------------------------------------------------------------------------------------
DEF  IS_MSG_ERR (iMsgNr:IN, iParam1:IN, iParam2:IN)
; Meldung die in allen Betriebsarten ausgegeben wird.
DECL INT iMsgNr
DECL INT MSG_QUIT_FLAG  ;Messages muessen quittiert werden.
DECL INT nHandle
DECL INT OFFSET
DECL STATE_T STATE
DECL CHAR MELDUNG[80]
DECL CHAR PARAM[10]
DECL INT IS_UserInstruction
CHAR ch_KXRKey[100]
CHAR ch_KXRKey_Btn1[10]
CHAR ch_KXRKey_Btn2[10]
DECL INT iParam1, iParam2
DECL KRLMSGPAR_T par1, par2

IS_UserInstruction=-1
;
IF IS_bHWCheckMode THEN
	RETURN
ENDIF
;
IF ($MODE_OP==#T1) OR ($MODE_OP==#T2) OR ((iMsgNr>=IS_IntErr_Param1) AND (iMsgNr<=IS_IntErr_Param6)) THEN
	MSG_QUIT_FLAG = 1
ELSE
	MSG_QUIT_FLAG = 2 ;Keine Quittierung in Automatik
ENDIF
;
;For Testing:
;MSG_QUIT_FLAG = 2
;
; Prepare the additional parameters
par1.par_type = #value
par2.par_type = #value
;
IF NOT (Varstate ("iParam1")==#initialized) then
   iParam1 = 0;
ENDIF
;
IF NOT (Varstate ("iParam2")==#initialized) then
   iParam2 = 0;
ENDIF
;
SWITCH iMsgNr
;Sync
CASE IS_MSG_ERR_SYNC1A
	ch_KXRKey[] = "IS_MSG_ERR_SYNC1A"
CASE IS_MSG_ERR_SYNC1B
	ch_KXRKey[] = "IS_MSG_ERR_SYNC1B"
	IS_UserInstruction = IS_Instr_Response
CASE IS_MSG_ERR_SYNC2A
	ch_KXRKey[] = "IS_MSG_ERR_SYNC2A"
CASE IS_MSG_ERR_SYNC2B
	ch_KXRKey[] = "IS_MSG_ERR_SYNC2B"
	IS_UserInstruction = IS_Instr_Response
;
;Select
CASE IS_MSG_ERR_SELECT1
	ch_KXRKey[] = "IS_MSG_ERR_SELECT1"
	IS_UserInstruction = IS_Instr_ModelCmp
CASE IS_MSG_ERR_SELECT1A
	ch_KXRKey[] = "IS_MSG_ERR_SELECT1A"
	IS_UserInstruction = IS_Instr_ModelChk
CASE IS_MSG_ERR_SELECT1B
	ch_KXRKey[] = "IS_MSG_ERR_SELECT1B"
	IS_UserInstruction = IS_Instr_DeadlyErr
CASE IS_MSG_ERR_SELECT1C
	ch_KXRKey[] = "IS_MSG_ERR_SELECT1C"
	IS_UserInstruction = IS_Instr_Response
CASE IS_MSG_ERR_SELECT2
	ch_KXRKey[] = "IS_MSG_ERR_SELECT2"
	IS_UserInstruction = IS_Instr_Response
CASE IS_MSG_ERR_SELECT2A
	ch_KXRKey[] = "IS_MSG_ERR_SELECT2A"
	IS_UserInstruction = IS_Instr_DeadlyErr
CASE IS_MSG_ERR_SELECT2B
	ch_KXRKey[] = "IS_MSG_ERR_SELECT2B"
CASE IS_MSG_ERR_SELECT3
	ch_KXRKey[] = "IS_MSG_ERR_SELECT3"
	IS_UserInstruction = IS_Instr_RoutCheck
CASE IS_MSG_ERR_SELECT3A
	ch_KXRKey[] = "IS_MSG_ERR_SELECT3A"
	IS_UserInstruction = IS_Instr_Response
;
;IMT Prepare
CASE IS_MSG_ERR_IMT_PREPARE1
	ch_KXRKey[] = "IS_MSG_ERR_IMT_PREPARE1"
CASE IS_MSG_ERR_IMT_PREPARE1A
	ch_KXRKey[] = "IS_MSG_ERR_IMT_PREPARE1A"
	IS_UserInstruction = IS_Instr_PntChk
CASE IS_MSG_ERR_IMT_PREPARE1B
	ch_KXRKey[] = "IS_MSG_ERR_IMT_PREPARE1B"
	IS_UserInstruction = IS_Instr_Response
;
;IMT_APPLY
CASE IS_MSG_ERR_IMT_APPLY
	ch_KXRKey[] = "IS_MSG_ERR_IMT_APPLY"
;
;Achsen senden
CASE IS_MSG_ERR_AXIS1
	ch_KXRKey[] = "IS_MSG_ERR_AXIS1"
CASE IS_MSG_ERR_AXIS1A
	ch_KXRKey[] = "IS_MSG_ERR_AXIS1A"
CASE IS_MSG_ERR_AXIS1B
	ch_KXRKey[] = "IS_MSG_ERR_AXIS1B"
CASE IS_MSG_ERR_AXIS1C
	ch_KXRKey[] = "IS_MSG_ERR_AXIS1C"
	IS_UserInstruction = IS_Instr_DeadlyErr
CASE IS_MSG_ERR_AXIS1D
	ch_KXRKey[] = "IS_MSG_ERR_AXIS1D"
	IS_UserInstruction = IS_Instr_Response
CASE IS_MSG_ERR_AXIS2
	ch_KXRKey[] = "IS_MSG_ERR_AXIS2"
	IS_UserInstruction = IS_Instr_DeadlyErr
CASE IS_MSG_ERR_AXIS2A
	ch_KXRKey[] = "IS_MSG_ERR_AXIS2A"
	IS_UserInstruction = IS_Instr_DeadlyErr
CASE IS_MSG_ERR_AXIS2B
	ch_KXRKey[] = "IS_MSG_ERR_AXIS2B"
	IS_UserInstruction = IS_Instr_Response
CASE IS_MSG_ERR_AXIS3
	ch_KXRKey[] = "IS_MSG_ERR_AXIS3"
	IS_UserInstruction = IS_Instr_DeadlyErr
CASE IS_MSG_ERR_AXIS3A
	ch_KXRKey[] = "IS_MSG_ERR_AXIS3A"
	IS_UserInstruction = IS_Instr_DeadlyErr
CASE IS_MSG_ERR_AXIS3B
	ch_KXRKey[] = "IS_MSG_ERR_AXIS3B"
	IS_UserInstruction = IS_Instr_Response
CASE IS_MSG_ERR_AXIS4
	ch_KXRKey[] = "IS_MSG_ERR_AXIS4"
	IS_UserInstruction = IS_Instr_DeadlyErr
CASE IS_MSG_ERR_AXIS4A
	ch_KXRKey[] = "IS_MSG_ERR_AXIS4A"
	IS_UserInstruction = IS_Instr_DeadlyErr
CASE IS_MSG_ERR_AXIS4B
	ch_KXRKey[] = "IS_MSG_ERR_AXIS4B"
	IS_UserInstruction = IS_Instr_Response
;
;Base senden
CASE IS_MSG_ERR_BASE1
	ch_KXRKey[] = "IS_MSG_ERR_BASE1"
	IS_UserInstruction = IS_Instr_DeadlyErr
CASE IS_MSG_ERR_BASE1A
	ch_KXRKey[] = "IS_MSG_ERR_BASE1A"
	IS_UserInstruction = IS_Instr_DeadlyErr
CASE IS_MSG_ERR_BASE1B
	ch_KXRKey[] = "IS_MSG_ERR_BASE2B"
	IS_UserInstruction = IS_Instr_Response
CASE IS_MSG_ERR_BASE2
	ch_KXRKey[] = "IS_MSG_ERR_BASE2"
	IS_UserInstruction = IS_Instr_DeadlyErr
CASE IS_MSG_ERR_BASE2A
	ch_KXRKey[] = "IS_MSG_ERR_BASE2A"
	IS_UserInstruction = IS_Instr_DeadlyErr
CASE IS_MSG_ERR_BASE2B
	ch_KXRKey[] = "IS_MSG_ERR_BASE2B"
	IS_UserInstruction = IS_Instr_Response
CASE IS_MSG_ERR_BASE3
	ch_KXRKey[] = "IS_MSG_ERR_BASE3"
	IS_UserInstruction = IS_Instr_DeadlyErr
CASE IS_MSG_ERR_BASE3A
	ch_KXRKey[] = "IS_MSG_ERR_BASE3A"
	IS_UserInstruction = IS_Instr_DeadlyErr
CASE IS_MSG_ERR_BASE3B
	ch_KXRKey[] = "IS_MSG_ERR_BASE3B"
	IS_UserInstruction = IS_Instr_Response
;
;IMT EndPose
CASE IS_MSG_ERR_IMT_END1
	ch_KXRKey[] = "IS_MSG_ERR_IMT_END1"
CASE IS_MSG_ERR_IMT_END1A
	ch_KXRKey[] = "IS_MSG_ERR_IMT_END1A"
CASE IS_MSG_ERR_IMT_END1B
	ch_KXRKey[] = "IS_MSG_ERR_IMT_END1B"
	IS_UserInstruction = IS_Instr_TolChk
CASE IS_MSG_ERR_IMT_END1C
	ch_KXRKey[] = "IS_MSG_ERR_IMT_END1C"
	IS_UserInstruction = IS_Instr_Response
;
;GetCorr
CASE IS_MSG_ERR_GETCORR1
	ch_KXRKey[] = "IS_MSG_ERR_GETCORR1"
	IS_UserInstruction = IS_Instr_DeadlyErr
CASE IS_MSG_ERR_GETCORR1A
	ch_KXRKey[] = "IS_MSG_ERR_GETCORR1A"
	IS_UserInstruction = IS_Instr_DeadlyErr
CASE IS_MSG_ERR_GETCORR1B
	ch_KXRKey[] = "IS_MSG_ERR_GETCORR1B"
	IS_UserInstruction = IS_Instr_Response
CASE IS_MSG_ERR_GETCORR2
	ch_KXRKey[] = "IS_MSG_ERR_GETCORR2"
	IS_UserInstruction = IS_Instr_DeadlyErr
CASE IS_MSG_ERR_GETCORR2A
	ch_KXRKey[] = "IS_MSG_ERR_GETCORR2A"
	IS_UserInstruction = IS_Instr_DeadlyErr
CASE IS_MSG_ERR_GETCORR2B
	ch_KXRKey[] = "IS_MSG_ERR_GETCORR2B"
	IS_UserInstruction = IS_Instr_Response
CASE IS_MSG_ERR_GETCORR3
	ch_KXRKey[] = "IS_MSG_ERR_GETCORR3"
	IS_UserInstruction = IS_Instr_DeadlyErr
CASE IS_MSG_ERR_GETCORR3A
	ch_KXRKey[] = "IS_MSG_ERR_GETCORR3A"
	IS_UserInstruction = IS_Instr_DeadlyErr
CASE IS_MSG_ERR_GETCORR3B
	ch_KXRKey[] = "IS_MSG_ERR_GETCORR3B"
	IS_UserInstruction = IS_Instr_Response
CASE IS_MSG_ERR_GETCORR4
	ch_KXRKey[] = "IS_MSG_ERR_GETCORR4"
	IS_UserInstruction = IS_Instr_DeadlyErr
CASE IS_MSG_ERR_GETCORR4A
	ch_KXRKey[] = "IS_MSG_ERR_GETCORR4A"
	IS_UserInstruction = IS_Instr_Response
;
CASE IS_MSG_ERR_TOL_EXCEEDED
	ch_KXRKey[] = "IS_MSG_ERR_TOL_EXCEEDED"
	IS_UserInstruction = IS_Instr_RobTol
;
;RF_Reset
CASE IS_MSG_ERR_RF_INIT1A
  ch_KXRKey[] = "IS_MSG_ERR_RF_INIT1A"
CASE IS_MSG_ERR_RF_INIT2A
  ch_KXRKey[] = "IS_MSG_ERR_RF_INIT2A"
;
;RF_Prepare
CASE IS_MSG_ERR_RF_PREPARE1
	ch_KXRKey[] = "IS_MSG_ERR_RF_PREPARE1"
	IS_UserInstruction = IS_Instr_DeadlyErr
CASE IS_MSG_ERR_RF_PREPARE1A
	ch_KXRKey[] = "IS_MSG_ERR_RF_PREPARE1A"
	IS_UserInstruction = IS_Instr_DeadlyErr
CASE IS_MSG_ERR_RF_PREPARE1B
	ch_KXRKey[] = "IS_MSG_ERR_RF_PREPARE1B"
	IS_UserInstruction = IS_Instr_Response
CASE IS_MSG_ERR_RF_PREPARE2
	ch_KXRKey[] = "IS_MSG_ERR_RF_PREPARE2"
	IS_UserInstruction = IS_Instr_DeadlyErr
CASE IS_MSG_ERR_RF_PREPARE2A
	ch_KXRKey[] = "IS_MSG_ERR_RF_PREPARE2A"
	IS_UserInstruction = IS_Instr_DeadlyErr
CASE IS_MSG_ERR_RF_PREPARE2B
	ch_KXRKey[] = "IS_MSG_ERR_RF_PREPARE2B"
	IS_UserInstruction = IS_Instr_Response
CASE IS_MSG_ERR_RF_PREPARE3
	ch_KXRKey[] = "IS_MSG_ERR_RF_PREPARE3"
	IS_UserInstruction = IS_Instr_DeadlyErr
CASE IS_MSG_ERR_RF_PREPARE3A
	ch_KXRKey[] = "IS_MSG_ERR_RF_PREPARE3A"
	IS_UserInstruction = IS_Instr_TypeChk
CASE IS_MSG_ERR_RF_PREPARE3B
	ch_KXRKey[] = "IS_MSG_ERR_RF_PREPARE3B"
	IS_UserInstruction = IS_Instr_DeadlyErr
CASE IS_MSG_ERR_RF_PREPARE3C
	ch_KXRKey[] = "IS_MSG_ERR_RF_PREPARE3C"
	IS_UserInstruction = IS_Instr_Response
;
;RF_APPLY
CASE IS_MSG_ERR_RF_APPLY1
	ch_KXRKey[] = "IS_MSG_ERR_RF_APPLY1"
	IS_UserInstruction = IS_Instr_DeadlyErr
;
CASE IS_MSG_ERR_RF_APPLY2
	ch_KXRKey[] = "IS_MSG_ERR_RF_APPLY2"
	IS_UserInstruction = IS_Instr_DeadlyErr
CASE IS_MSG_ERR_RF_APPLY2A
	ch_KXRKey[] = "IS_MSG_ERR_RF_APPLY2A"
	IS_UserInstruction = IS_Instr_Response
CASE IS_MSG_ERR_RF_APPLY2B
	ch_KXRKey[] = "IS_MSG_ERR_RF_APPLY2B"
	IS_UserInstruction = IS_Instr_DeadlyErr
;
CASE IS_MSG_ERR_RF_APPLY3
	ch_KXRKey[] = "IS_MSG_ERR_RF_APPLY3"
	IS_UserInstruction = IS_Instr_DeadlyErr
CASE IS_MSG_ERR_RF_APPLY3A
	ch_KXRKey[] = "IS_MSG_ERR_RF_APPLY3A"
	IS_UserInstruction = IS_Instr_Response
CASE IS_MSG_ERR_RF_APPLY3B
	ch_KXRKey[] = "IS_MSG_ERR_RF_APPLY3B"
	IS_UserInstruction = IS_Instr_ImgMsgChk
CASE IS_MSG_ERR_RF_APPLY3C
	ch_KXRKey[] = "IS_MSG_ERR_RF_APPLY3C"
	IS_UserInstruction = IS_Instr_ImgMsgChk
CASE IS_MSG_ERR_RF_APPLY3D
	ch_KXRKey[] = "IS_MSG_ERR_RF_APPLY3D"
	IS_UserInstruction = IS_Instr_TolChk
CASE IS_MSG_ERR_RF_APPLY3E
	ch_KXRKey[] = "IS_MSG_ERR_RF_APPLY3E"
	IS_UserInstruction = IS_Instr_HWChk
;
CASE IS_MSG_ERR_RF_APPLY4
	ch_KXRKey[] = "IS_MSG_ERR_RF_APPLY4"
	IS_UserInstruction = IS_Instr_DeadlyErr
CASE IS_MSG_ERR_RF_APPLY4A
	ch_KXRKey[] = "IS_MSG_ERR_RF_APPLY4A"
	IS_UserInstruction = IS_Instr_Response
CASE IS_MSG_ERR_RF_APPLY4B
	ch_KXRKey[] = "IS_MSG_ERR_RF_APPLY4B"
	IS_UserInstruction = IS_Instr_DeadlyErr
CASE IS_MSG_ERR_RF_APPLY4C
	ch_KXRKey[] = "IS_MSG_ERR_RF_APPLY4C"
	IS_UserInstruction = IS_Instr_ImgMsgChk
CASE IS_MSG_ERR_RF_APPLY4D
	ch_KXRKey[] = "IS_MSG_ERR_RF_APPLY4D"
	IS_UserInstruction = IS_Instr_TolChk
CASE IS_MSG_ERR_RF_APPLY4E
	ch_KXRKey[] = "IS_MSG_ERR_RF_APPLY4E"
	IS_UserInstruction = IS_Instr_HWChk
;
CASE IS_MSG_ERR_RF_APPLY5
	ch_KXRKey[] = "IS_MSG_ERR_RF_APPLY5"
	IS_UserInstruction = IS_Instr_DeadlyErr
CASE IS_MSG_ERR_RF_APPLY5A
	ch_KXRKey[] = "IS_MSG_ERR_RF_APPLY5A"
	IS_UserInstruction = IS_Instr_Response
CASE IS_MSG_ERR_RF_APPLY5B
	ch_KXRKey[] = "IS_MSG_ERR_RF_APPLY5B"
	IS_UserInstruction = IS_Instr_ImgMsgChk
CASE IS_MSG_ERR_RF_APPLY5C
	ch_KXRKey[] = "IS_MSG_ERR_RF_APPLY5C"
	IS_UserInstruction = IS_Instr_ImgMsgChk
CASE IS_MSG_ERR_RF_APPLY5D
	ch_KXRKey[] = "IS_MSG_ERR_RF_APPLY5D"
	IS_UserInstruction = IS_Instr_TolChk
CASE IS_MSG_ERR_RF_APPLY5E
	ch_KXRKey[] = "IS_MSG_ERR_RF_APPLY5E"
	IS_UserInstruction = IS_Instr_HWChk
;
CASE IS_MSG_ERR_RF_APPLY6
	ch_KXRKey[] = "IS_MSG_ERR_RF_APPLY6"
	IS_UserInstruction = IS_Instr_DeadlyErr
;
;RF_ENDPOSE
CASE IS_MSG_ERR_RF_END1
	ch_KXRKey[] = "IS_MSG_ERR_RF_END1"
	IS_UserInstruction = IS_Instr_DeadlyErr
CASE IS_MSG_ERR_RF_END1A
	ch_KXRKey[] = "IS_MSG_ERR_RF_END1A"
	IS_UserInstruction = IS_Instr_MsgChk
CASE IS_MSG_ERR_RF_END1B
	ch_KXRKey[] = "IS_MSG_ERR_RF_END1B"
	IS_UserInstruction = IS_Instr_ImgMsgChk
CASE IS_MSG_ERR_RF_END1C
	ch_KXRKey[] = "IS_MSG_ERR_RF_END1C"
	IS_UserInstruction = IS_Instr_TolChk
CASE IS_MSG_ERR_RF_END1D
	ch_KXRKey[] = "IS_MSG_ERR_RF_END1D"
	IS_UserInstruction = IS_Instr_Response
CASE IS_MSG_ERR_RF_END1E
  ch_KXRKey[] = "IS_MSG_ERR_RF_END1E"
  IS_UserInstruction = IS_Instr_HWChk
;
CASE IS_MSG_ERR_RF_END2
	ch_KXRKey[] = "IS_MSG_ERR_RF_END2"
	IS_UserInstruction = IS_Instr_DeadlyErr
CASE IS_MSG_ERR_RF_END2A
	ch_KXRKey[] = "IS_MSG_ERR_RF_END2A"
	IS_UserInstruction = IS_Instr_MsgChk
CASE IS_MSG_ERR_RF_END2B
	ch_KXRKey[] = "IS_MSG_ERR_RF_END2B"
	IS_UserInstruction = IS_Instr_MsgChk
CASE IS_MSG_ERR_RF_END2C
	ch_KXRKey[] = "IS_MSG_ERR_RF_END2C"
	IS_UserInstruction = IS_Instr_TolChk
CASE IS_MSG_ERR_RF_END2D
	ch_KXRKey[] = "IS_MSG_ERR_RF_END2D"
	IS_UserInstruction = IS_Instr_Response
CASE IS_MSG_ERR_RF_END2E
  ch_KXRKey[] = "IS_MSG_ERR_RF_END2E"
  IS_UserInstruction = IS_Instr_HWChk
;
CASE IS_MSG_ERR_RF_END3
	ch_KXRKey[] = "IS_MSG_ERR_RF_END3"
	IS_UserInstruction = IS_Instr_RobProg
;
;RF_GETCORRECTION
CASE IS_MSG_ERR_RF_CORR1
  ch_KXRKey[] = "IS_MSG_ERR_RF_CORR1"
  IS_UserInstruction = IS_Instr_DeadlyErr
CASE IS_MSG_ERR_RF_CORR1A
  ch_KXRKey[] = "IS_MSG_ERR_RF_CORR1A"
  IS_UserInstruction = IS_Instr_Response
CASE IS_MSG_ERR_RF_CORR1B
  ch_KXRKey[] = "IS_MSG_ERR_RF_CORR1B"
CASE IS_MSG_ERR_RF_CORR2
  ch_KXRKey[] = "IS_MSG_ERR_RF_CORR2"
  IS_UserInstruction = IS_Instr_DeadlyErr
CASE IS_MSG_ERR_RF_CORR2A
  ch_KXRKey[] = "IS_MSG_ERR_RF_CORR2A"
  IS_UserInstruction = IS_Instr_Response
CASE IS_MSG_ERR_RF_CORR2B
  ch_KXRKey[] = "IS_MSG_ERR_RF_CORR2B"
CASE IS_MSG_ERR_RF_CORR3
  ch_KXRKey[] = "IS_MSG_ERR_RF_CORR3"
;
;Service
CASE IS_MSG_ERR_SERV_SENS1
	ch_KXRKey[] = "IS_MSG_ERR_SERV_SENS1"
	IS_UserInstruction = 0
	IS_Apply_Service(3) ;3
CASE IS_MSG_ERR_SERV_SENS2
	ch_KXRKey[] = "IS_MSG_ERR_SERV_SENS2"
	IS_UserInstruction = 0
CASE IS_MSG_ERR_SERV_TOOL
	ch_KXRKey[] = "IS_MSG_ERR_SERV_TOOL"
	IS_UserInstruction = 0
CASE IS_MSG_ERR_SERV_TOOL_T
	ch_KXRKey[] = "IS_MSG_ERR_SERV_TOOL_T"
	IS_UserInstruction = IS_Instr_TolChk
CASE IS_MSG_ERR_SERV_ROB
	ch_KXRKey[] = "IS_MSG_ERR_SERV_ROB"
	IS_UserInstruction = 0
CASE IS_MSG_ERR_SERV_ROB_T
	ch_KXRKey[] = "IS_MSG_ERR_SERV_ROB_T"
	IS_UserInstruction = IS_Instr_TolChk
CASE IS_MSG_ERR_SERV_SENSIMT
	ch_KXRKey[] = "IS_MSG_ERR_SERV_SENSIMT"
CASE IS_MSG_ERR_SERVICE1A
	ch_KXRKey[] = "IS_MSG_ERR_SERVICE1A"
	IS_UserInstruction = IS_Instr_Response
CASE IS_MSG_ERR_SERVICE1B
	ch_KXRKey[] = "IS_MSG_ERR_SERVICE1B"
	IS_UserInstruction = IS_Instr_Response
CASE IS_MSG_ERR_SERVICE1C
	ch_KXRKey[] = "IS_MSG_ERR_SERVICE1C"
	IS_UserInstruction = IS_Instr_Response
CASE IS_MSG_ERR_SERVICE1D
	ch_KXRKey[] = "IS_MSG_ERR_SERVICE1D"
	IS_UserInstruction = IS_Instr_Response
CASE IS_MSG_ERR_SERVICE1E
	ch_KXRKey[] = "IS_MSG_ERR_SERVICE1E"
CASE IS_MSG_ERR_SERVICE1F
	ch_KXRKey[] = "IS_MSG_ERR_SERVICE1F"
CASE IS_MSG_ERR_SERVICE1G
	ch_KXRKey[] = "IS_MSG_ERR_SERVICE1G"
CASE IS_MSG_ERR_SERVICE1H
	ch_KXRKey[] = "IS_MSG_ERR_SERVICE1H"
;
CASE IS_MSG_ERR_RTC
	ch_KXRKey[] = "IS_MSG_ERR_RTC"
	IS_UserInstruction = IS_Instr_CalChk
CASE IS_MSG_ERR_RTC_CALIB
	ch_KXRKey[] = "IS_MSG_ERR_RTC_CALIB"
CASE IS_MSG_ERR_RTC_CALC_TOOL
	ch_KXRKey[] = "IS_MSG_ERR_RTC_CALC_TOOL"
CASE IS_MSG_ERR_RTC_CALC_BASE
	ch_KXRKey[] = "IS_MSG_ERR_RTC_CALC_BASE"
CASE IS_MSG_ERR_REQUEST
	ch_KXRKey[] = "IS_MSG_ERR_REQUEST"
CASE IS_MSG_ERR_BASE
	ch_KXRKey[] = "IS_MSG_ERR_BASE"
CASE IS_MSG_ERR_BIT_TRNS
	ch_KXRKey[] = "IS_MSG_ERR_BIT_TRNS"
CASE IS_MSG_ERR_TRANSM
	ch_KXRKey[] = "IS_MSG_ERR_TRANSM"
CASE IS_MSG_PP_WARN
	ch_KXRKey[] = "IS_MSG_PP_WARN"
CASE IS_MSG_PP_MOVEMODE
	ch_KXRKey[] = "IS_MSG_PP_MOVEMODE"
CASE IS_MSG_PP_TOL
	ch_KXRKey[] = "IS_MSG_PP_TOL"
CASE IS_MSG_PP_INVERSE
	ch_KXRKey[] = "IS_MSG_PP_INVERSE"
CASE IS_MSG_PP_FORWARD
	ch_KXRKey[] = "IS_MSG_PP_FORWARD"
CASE IS_MSG_PP_TEST_POSA
	ch_KXRKey[] = "IS_MSG_PP_TEST_POSA"
CASE IS_MSG_PP_TEST_POSK
	ch_KXRKey[] = "IS_MSG_PP_TEST_POSK"
CASE IS_MSG_DEBUG
	ch_KXRKey[] = "IS_MSG_DEBUG"
;
;Zustand/Warnung
CASE IS_MSG_RESULT_OK
  ch_KXRKey[] = "IS_MSG_RESULT_OK"
CASE IS_MSG_RESULT_NOK
  ch_KXRKey[] = "IS_MSG_RESULT_NOK"
CASE IS_MSG_WARN_TOL
  ch_KXRKey[] = "IS_MSG_WARN_TOL"
;
; Fehler und Meldungen von intern
CASE IS_IntErr_Param1
  ch_KXRKey[] = "IS_IntErr_Param1"
CASE IS_IntErr_Param2
  ch_KXRKey[] = "IS_IntErr_Param2"
CASE IS_IntErr_Param3
  ch_KXRKey[] = "IS_IntErr_Param3"
CASE IS_IntErr_Param4
  ch_KXRKey[] = "IS_IntErr_Param4"
CASE IS_IntErr_Param5
  ch_KXRKey[] = "IS_IntErr_Param5"
CASE IS_IntErr_Param6
  ch_KXRKey[] = "IS_IntErr_Param6"
;
CASE IS_IntErr_Com
	ch_KXRKey[] = "IS_IntErr_Com"
CASE IS_IntErr_ERequest
 ch_KXRKey[] = "IS_IntErr_ERequest"
CASE IS_IntErr_Meas
  ch_KXRKey[] = "IS_IntErr_Meas"
CASE IS_IntErr_Retry
  ch_KXRKey[] = "IS_IntErr_Retry"
CASE IS_IntErr_Data
  ch_KXRKey[] = "IS_IntErr_Data"
CASE IS_IntErr_Base
  ch_KXRKey[] = "IS_IntErr_Base"
CASE IS_IntErr_Tool
  ch_KXRKey[] = "IS_IntErr_Tool"
CASE IS_IntErr_ESendBit
 ch_KXRKey[] = "IS_IntErr_ESendBit"
CASE IS_IntErr_Specif
  ch_KXRKey[] = "IS_IntErr_Specif"
CASE IS_IntErr_SrvcExp
 	ch_KXRKey[] = "IS_IntErr_SrvcExp"
CASE IS_IntErr_StReq1
  ch_KXRKey[] = "IS_IntErr_StReq1"
CASE IS_IntErr_StReq2
  ch_KXRKey[] = "IS_IntErr_StReq2"
CASE IS_IntErr_ESend
 	ch_KXRKey[] = "IS_IntErr_ESend"
CASE IS_IntErr_IQRWait
 	ch_KXRKey[] = "IS_IntErr_IQRWait"
 	MSG_QUIT_FLAG = 3
CASE IS_IntErr_PCWait
 	ch_KXRKey[] = "IS_IntErr_PCWait"
 	MSG_QUIT_FLAG = 3
CASE IS_IntErr_TolRob
 	ch_KXRKey[] = "IS_IntErr_TolRob"
CASE IS_IntErr_RFAState
  ch_KXRKey[] = "IS_IntErr_RFAState"
CASE IS_IntErr_MeasPosNo
  ch_KXRKey[] = "IS_IntErr_MeasPosNo"
CASE IS_IntErr_RFGCSt
	ch_KXRKey[] = "IS_IntErr_RFGCSt"
CASE IS_IntErr_RFEPSt
	ch_KXRKey[] = "IS_IntErr_RFEPSt"
;
DEFAULT
   ch_KXRKey[] = "IS_MSG_ERR_DEFAULT"
ENDSWITCH
;
;Set Parameters:
par1.par_int = iParam1
par2.par_int = iParam2
;
SWITCH MSG_QUIT_FLAG
CASE 1
	IF (iMsgNr == IS_IntErr_Com) THEN
		;Dauerschleife bis Verbindung wieder da ist und der Ablauf normal weiter geht oder Option zum simulieren:
		IS_RF_ReconnectLoop()
	ELSE
 		OFFSET = 0
 		;
 		;Liegt eine Handlungsanweisung vor?
 		IF (IS_UserInstruction <> -1) THEN
	 	  REPEAT
	 	  	; Solange wiederholen bis Dialog mit OK/Weiter bestätigt wird.
	 	  	IF (IS_iServiceMode == IS_iSERVICE_NONE) THEN
	 	  		; Wenn nicht in Serviceprogramm, dann Button Info&Weiter, da Frage nach Messwiederholung folgt
	 	  		ch_KXRKey_Btn1[]="INFO"
					ch_KXRKey_Btn2[]="FORWARD"
	 	  		IS_ShowDialog(IS_ANSWER,ch_KXRKey_Btn1[],ch_KXRKey_Btn2[]," "," "," "," "," ",ch_KXRKey[], "vw_isr_usr_r", TRUE, par1, par2)
	 	  	ELSE
	 	  		; Wenn in Serviceprogramm, dann Button Info&OK
	 	  		ch_KXRKey_Btn1[]="INFO"
					ch_KXRKey_Btn2[]="OK"
	 	  		IS_ShowDialog(IS_ANSWER,ch_KXRKey_Btn1[],ch_KXRKey_Btn2[]," "," "," "," "," ",ch_KXRKey[], "vw_isr_usr_r", TRUE, par1, par2)
	 	  	ENDIF
		 		IS_ANSWER = 8-IS_ANSWER
				IF (IS_ANSWER == 1) THEN
					;'Info': Handlungsanweisung anzeigen
					IS_GetUserInstruction(IS_UserInstruction)
				ELSE
					;'OK': Beenden ohne Handlungsanweisung
				ENDIF
			UNTIL (IS_ANSWER <> 1)
 		ELSE
 			; Dialog ohne Info-Button anzeigen
 			ch_KXRKey_Btn2[]="OK"
 			IS_ShowDialog(IS_ANSWER," ",ch_KXRKey_Btn2[]," "," "," "," "," ",ch_KXRKey[], "vw_isr_usr_r", TRUE, par1, par2)
 		ENDIF
	ENDIF
CASE 2
  IS_ShowMessage(nHandle, #notify, ch_KXRKey[], "vw_isr_usr_r", iMsgNr, TRUE, par1, par2)
ENDSWITCH
;
END ;of IS_MSG_ERR
;---------------------------------------------------------------------------------------------
;ENDFOLD
;
;FOLD Meldungsausgabe (Info, Quittierung und Dialog)
;---------------------------------------------------------------------------------------------
DEF  IS_MSG(iMsgNr: IN, iMsgType: IN, iParam: IN)
DECL INT iMsgNr, iMsgType, iParam
DECL KRLMSGPAR_T par1
DECL INT nHandle
CHAR ch_KXRKey[100]
CHAR ch_KXRKey_btn1[10]
CHAR ch_KXRKey_btn2[10]
;
; Prepare the additional parameter
par1.par_type = #value

IF NOT (Varstate ("iParam")==#initialized) then
   iParam = 0;
ENDIF
;
IF (($MODE_OP==#T2) OR ($MODE_OP==#T1) OR (IS_iServiceMode <> IS_iSERVICE_NONE)) THEN
	SWITCH iMsgNr
	CASE IS_MSG_I_SERV_SENS_CHK
 	  ch_KXRKey[] = "IS_Info_Serv_Sens_Chk"
 	CASE IS_MSG_I_SERV_SENS
 		ch_KXRKey[] = "IS_Info_Serv_Sens"
 	CASE IS_MSG_I_SERV_TOOL
		ch_KXRKey[] = "IS_Info_Serv_Tool"
 	CASE IS_MSG_I_SERV_TOOL_PATH1
 		ch_KXRKey[] = "IS_Info_Serv_Tool_Path"
 	CASE IS_MSG_I_SERV_ROB
 	  ch_KXRKey[] = "IS_Info_Serv_Rob"
 	CASE IS_MSG_I_SERV_ROB_PATH1
 	  ch_KXRKey[] = "IS_Info_Serv_Rob_Path"
 	CASE IS_MSG_I_SERV_SENSIMT
 		ch_KXRKey[] = "IS_Info_Serv_Sens_IMT"
 	CASE IS_MSG_I_TRANS_AXES
 		ch_KXRKey[] = "IS_Info_Transfer_Axes"
	CASE IS_MSG_I_TRANS_BASE
		ch_KXRKey[] = "IS_Info_Transfer_Base"
	CASE IS_MSG_I_SYS_DIAG_1
		ch_KXRKey[] = "IS_Info_Sys_Diag_1"
	CASE IS_MSG_I_SYS_DIAG_2
		ch_KXRKey[] = "IS_Info_Sys_Diag_2"
	CASE IS_MSG_I_SYS_DIAG_3
		ch_KXRKey[] = "IS_Info_Sys_Diag_3"
	CASE IS_MSG_I_SYS_DIAG_4
		ch_KXRKey[] = "IS_Info_Sys_Diag_4"
	CASE IS_MSG_I_SYS_DIAG_5
		ch_KXRKey[] = "IS_Info_Sys_Diag_5"
  CASE IS_MSG_I_SYS_DIAG_6
		ch_KXRKey[] = "IS_Info_Sys_Diag_6"
	CASE IS_MSG_I_SYS_DIAG_7
 		ch_KXRKey[] = "IS_Info_Sys_Diag_7"
	CASE IS_MSG_I_SYNC
	  IF (IS_SYS_TYPE == IS_SYS_TYPE_IMT) THEN
	  	ch_KXRKey[] = "IS_Info_Sync_IMT"
	  ENDIF
	  IF (IS_SYS_TYPE == IS_SYS_TYPE_RF) THEN
	  	ch_KXRKey[] = "IS_Info_Sync_RF"
	  ENDIF
		ch_KXRKey_btn1[]= "YES"
		ch_KXRKey_btn2[]= "NO"
	CASE IS_MSG_I_MEAS_FAILED
	  IF (IS_SYS_TYPE == IS_SYS_TYPE_RF) THEN
			ch_KXRKey[] = "IS_Info_Meas_Failed"
			ch_KXRKey_btn1[]= "REPEAT"
			ch_KXRKey_btn2[]= "CANCEL"
		ENDIF
	CASE IS_MSG_I_SERV_TOOL_PATH2
	  IF (IS_SYS_TYPE == IS_SYS_TYPE_RF) THEN
			ch_KXRKey_btn1[]= "OK"
			ch_KXRKey_btn2[]= " "
			ch_KXRKey[] = "IS_Info_Tool_Path_2"
	  ENDIF
	CASE IS_MSG_I_SERV_ROB_PATH2
	  IF (IS_SYS_TYPE == IS_SYS_TYPE_RF) THEN
			ch_KXRKey_btn1[]= "OK"
			ch_KXRKey_btn2[]= " "
			ch_KXRKey[] = "IS_Info_Tool_Path_2"
	  ENDIF
	ENDSWITCH
	;
	; Set parameter
	par1.par_int = iParam
	;
	SWITCH iMsgType
		CASE IS_MSG_TYPE_DIALOG
			IS_ShowDialog(IS_ANSWER,ch_KXRKey_btn1[],ch_KXRKey_btn2[]," "," "," "," "," ",ch_KXRKey[], "vw_isr_usr_r", TRUE, par1)
			IS_ANSWER = 8-IS_ANSWER
		CASE IS_MSG_TYPE_NOTIFY
			IS_ShowMessage(nHandle, #notify, ch_KXRKey[], "vw_isr_usr_r", iMsgNr, TRUE, par1)
		CASE IS_MSG_TYPE_QUIT
			IS_ShowMessage(nHandle, #quit, ch_KXRKey[], "vw_isr_usr_r", iMsgNr, TRUE, par1)
		CASE IS_MSG_TYPE_STATE
			IS_ShowMessage(nHandle, #state, ch_KXRKey[], "vw_isr_usr_r", iMsgNr, TRUE, par1)
		DEFAULT
			IS_ShowMessage(nHandle, #notify, ch_KXRKey[], "vw_isr_usr_r", iMsgNr, TRUE, par1)
	ENDSWITCH
ENDIF
;
END ;of IS_MSG
;---------------------------------------------------------------------------------------------
;ENDFOLD
;
;FOLD Framemessage
;---------------------------------------------------------------------------------------------
DEF IS_MSG_FRAME2 (TYPE:IN, NR:IN, INFRAME:IN)
DECL FRAME INFRAME
DECL INT TYPE, NR
DECL INT OFFSET
DECL STATE_T STATE
DECL INT nHandle
DECL CHAR NAME[20]
DECL CHAR MELDUNG[80]
DECL CHAR ch_KXRkey[100]
DECL CHAR ABS[20]
;
SWITCH TYPE
  CASE 1
    NAME[]="Baseoffset"
    ABS[]="Differenz Basedaten"
  CASE 2
    NAME[]="Tooloffset"
    ABS[]="Differenz Tooldaten"
  CASE 3	;
    NAME[]="Base"
    ABS[]="Alte Basedaten"
  CASE 4
    NAME[]="Base"
    ABS[]="Neue Basedaten"
  CASE 5
    NAME[]="Tool"
    ABS[]="Alte Tooldaten"
  CASE 6
    NAME[]="Tool"
    ABS[]="Neue Tooldaten"
  CASE 7
    NAME[]="Base"
    ABS[]="Korrekturdaten"
  CASE 8
    NAME[]="Tool"
    ABS[]="Korrekturdaten"
  CASE 9
    NAME[]="Grenzwert"
    ABS[]="Korrekturdaten"
ENDSWITCH
;
	OFFSET=0
	IF (NR>0) THEN
  	SWRITE(MELDUNG[],STATE,OFFSET,"%s%d: X:%.1f,Y:%.1f,Z:%.1f,A:%.3f,B:%.3f,C:%.3f",NAME[],NR,INFRAME.x,INFRAME.y,INFRAME.z,INFRAME.a,INFRAME.b,INFRAME.c)
  	;SWRITE(MELDUNG[],STATE,OFFSET,"X:%.1f,Y:%.1f,Z:%.1f,A:%.3f,B:%.3f,C:%.3f",INFRAME.x,INFRAME.y,INFRAME.z,INFRAME.a,INFRAME.b,INFRAME.c)
  ELSE
  	SWRITE(MELDUNG[],STATE,OFFSET,"%s: X:%.1f,Y:%.1f,Z:%.1f,A:%.3f,B:%.3f,C:%.3f",NAME[],INFRAME.x,INFRAME.y,INFRAME.z,INFRAME.a,INFRAME.b,INFRAME.c)
 	ENDIF
;
  ;MsgState(nHandle, MELDUNG[], ABS[])
  IS_ShowMessage(nHandle, #state, MELDUNG[], ABS[], 1, TRUE)
;
END ;of IS_MSG_FRAME2()
;---------------------------------------------------------------------------------------------
;ENDFOLD
;
;FOLD ShowDialog
DEF IS_ShowDialog(nAnswer:OUT, sDialogSK1[]:IN,sDialogSK2[]:IN,sDialogSK3[]:IN,sDialogSK4[]:IN,sDialogSK5[]:IN,sDialogSK6[]:IN,sDialogSK7[]:IN,sText[]:IN, sModul[]:IN, bLog:IN, Par1:IN,Par2:IN,Par3:IN)
;************************************************************
;Function: Executes a dialog
;************************************************************
DECL KrlMsg_T Msg
DECL KrlMsgDlgSK_T Msg_SOFTKEY[7]
DECL INT nHandle,nMsgSel,nApplNum,nMsgTNr,count, len, nAnswer, nMsgNr
DECL BOOL bLog,Clear
DECL KrlMsgPar_T Par1,Par2,Par3, MsgPar[3]
DECL EKrlMsgType MsgType
DECL KrlMsgOpt_T MsgOpt
DECL CHAR sModul[], sText[], sDialogSK1[], sDialogSK2[], sDialogSK3[], sDialogSK4[], sDialogSK5[], sDialogSK6[], sDialogSK7[]

;set Parameter (if existent (otherwise "empty"))
ERR_CLEAR($Err)
ON_ERROR_PROCEED
MsgPar[1]=Par1
IF ($Err.Number<>0)THEN
  MsgPar[1].par_type=#empty
ENDIF
ERR_CLEAR($Err)
ON_ERROR_PROCEED
MsgPar[2]=Par2
IF ($Err.Number<>0)THEN
  MsgPar[2].par_type=#empty
ENDIF
ERR_CLEAR($Err)
ON_ERROR_PROCEED
MsgPar[3]=Par3
IF ($Err.Number<>0)THEN
  MsgPar[3].par_type=#empty
ENDIF

;set Option
;Vorlaufstopp
MsgOpt.Vl_Stop=FALSE
;Clear message on program reset
MsgOpt.Clear_P_Reset=TRUE
;Clear message on block selection
MsgOpt.Clear_p_SAW=FALSE
;Log message
MsgOpt.Log_To_DB=bLog

;Standard aus MSGLIB
Msg.Nr=1
ERR_CLEAR($Err)
ON_ERROR_PROCEED
Msg.Nr=nMsgNr
len=Strlen(sText[])
IF len>0 THEN
  IF len>80 THEN
    len=80
  ENDIF
  FOR count=1 TO len
    Msg.Msg_txt[count]=sText[count]
  ENDFOR
ELSE
  Msg.Msg_txt[]="parameter sText[] is missing"
ENDIF

len=Strlen(sModul[])
IF len>0 THEN
  IF len>24 THEN
    len=24
  ENDIF
  FOR count=1 TO len
    Msg.Modul[count]=sModul[count]
  ENDFOR
ELSE
  Msg.Modul[]="Appl"
ENDIF

;Set softkey text (1)
ERR_CLEAR($Err)
ON_ERROR_PROCEED
len=Strlen(sDialogSK1[])
IF $Err.Number==0 THEN
  IF len > 0 THEN
    IF len>24 THEN
      len=24
    ENDIF
    Msg_SOFTKEY[7].Sk_Type = #KEY
    FOR count=1 TO len
      Msg_SOFTKEY[7].Sk_txt[count] = sDialogSK1[count]
    ENDFOR
  ENDIF
ELSE
  FOR count=1 TO 24
    Msg_SOFTKEY[7].Sk_txt[count] = " "
  ENDFOR
ENDIF

;Set softkey text (2)
ERR_CLEAR($Err)
ON_ERROR_PROCEED
len=Strlen(sDialogSK2[])
IF $Err.Number==0 THEN
  len=Strlen(sDialogSK2[])
  IF len > 0 THEN
    IF len>24 THEN
      len=24
    ENDIF
    Msg_SOFTKEY[6].Sk_Type = #KEY
    FOR count=1 TO len
      Msg_SOFTKEY[6].Sk_txt[count] = sDialogSK2[count]
    ENDFOR
  ENDIF
ELSE
  FOR count=1 TO 24
    Msg_SOFTKEY[6].Sk_txt[count] = " "
  ENDFOR
ENDIF

;Set softkey text (3)
ERR_CLEAR($Err)
ON_ERROR_PROCEED
len=Strlen(sDialogSK3[])
IF $Err.Number==0 THEN
  len=Strlen(sDialogSK3[])
  IF len > 0 THEN
    IF len>24 THEN
      len=24
    ENDIF
    Msg_SOFTKEY[5].Sk_Type = #KEY
    FOR count=1 TO len
      Msg_SOFTKEY[5].Sk_txt[count] = sDialogSK3[count]
    ENDFOR
  ENDIF
ELSE
  FOR count=1 TO 24
    Msg_SOFTKEY[5].Sk_txt[count] = " "
  ENDFOR
ENDIF

;Set softkey text (4)
ERR_CLEAR($Err)
ON_ERROR_PROCEED
len=Strlen(sDialogSK4[])
IF $Err.Number==0 THEN
  len=Strlen(sDialogSK4[])
  IF len > 0 THEN
    IF len>24 THEN
      len=24
    ENDIF
    Msg_SOFTKEY[4].Sk_Type = #KEY
    FOR count=1 TO len
      Msg_SOFTKEY[4].Sk_txt[count] = sDialogSK4[count]
    ENDFOR
  ENDIF
ELSE
  FOR count=1 TO 24
    Msg_SOFTKEY[4].Sk_txt[count] = " "
  ENDFOR
ENDIF

;Set softkey text (5)
ERR_CLEAR($Err)
ON_ERROR_PROCEED
len=Strlen(sDialogSK5[])
IF $Err.Number==0 THEN
  len=Strlen(sDialogSK5[])
  IF len > 0 THEN
    IF len>24 THEN
      len=24
    ENDIF
    Msg_SOFTKEY[3].Sk_Type = #KEY
    FOR count=1 TO len
      Msg_SOFTKEY[3].Sk_txt[count] = sDialogSK5[count]
    ENDFOR
  ENDIF
ELSE
  FOR count=1 TO 24
    Msg_SOFTKEY[3].Sk_txt[count] = " "
  ENDFOR
ENDIF

;Set softkey text (6)
ERR_CLEAR($Err)
ON_ERROR_PROCEED
len=Strlen(sDialogSK6[])
IF $Err.Number==0 THEN
  len=Strlen(sDialogSK6[])
  IF len > 0 THEN
    IF len>24 THEN
      len=24
    ENDIF
    Msg_SOFTKEY[2].Sk_Type = #KEY
    FOR count=1 TO len
      Msg_SOFTKEY[2].Sk_txt[count] = sDialogSK6[count]
    ENDFOR
  ENDIF
ELSE
  FOR count=1 TO 24
    Msg_SOFTKEY[2].Sk_txt[count] = " "
  ENDFOR
ENDIF

;Set softkey text (7)
ERR_CLEAR($Err)
ON_ERROR_PROCEED
len=Strlen(sDialogSK7[])
IF $Err.Number==0 THEN
  len=Strlen(sDialogSK7[])
  IF len > 0 THEN
    IF len>24 THEN
      len=24
    ENDIF
    Msg_SOFTKEY[1].Sk_Type = #KEY
    FOR count=1 TO len
      Msg_SOFTKEY[1].Sk_txt[count] = sDialogSK7[count]
    ENDFOR
  ENDIF
ELSE
  FOR count=1 TO 24
    Msg_SOFTKEY[1].Sk_txt[count] = " "
  ENDFOR
ENDIF

CONTINUE
nHandle=SET_KRLDLG(Msg, MsgPar[], Msg_SOFTKEY[], MsgOpt)

If (nHandle > 0) THEN
  REPEAT
  CONTINUE
  WAIT SEC 0.5
  UNTIL((NOT Exists_KrlDlg(nHandle, nAnswer)))
  Clear=Clear_KrlMsg(nHANDLE)
ENDIF
;
END
;
;
DEF IS_ShowMessage(nHandle:OUT, MsgType:IN, sText[]:IN, sModul[]:IN, nMsgNr:IN, bLog:IN, Par1:IN, Par2:IN, Par3:IN)
;************************************************************
;Function: Executes a Message Send of the notify message
;************************************************************
DECL CHAR sText[], sModul[]
DECL KrlMsg_T Msg
DECL EKrlMsgType MsgType
DECL KrlMsgPar_T Par1, Par2, Par3, MsgPar[3]
DECL KrlMsgOpt_T MsgOpt
DECL BOOL bLog
DECL INT count, len, nHandle, nMsgNr

;set Parameter (if existent (otherwise "empty"))
ERR_CLEAR($Err)
ON_ERROR_PROCEED
MsgPar[1]=Par1
if ($Err.Number<>0)Then
  MsgPar[1].par_type=#empty
endif
ERR_CLEAR($Err)
ON_ERROR_PROCEED
  MsgPar[2]=Par2
if ($Err.Number<>0)Then
MsgPar[2].par_type=#empty
endif
ERR_CLEAR($Err)
ON_ERROR_PROCEED
  MsgPar[3]=Par3
if ($Err.Number<>0)Then
  MsgPar[3].par_type=#empty
endif

;set Option
;Vorlaufstopp
MsgOpt.Vl_Stop=FALSE
;Clear message on program reset
MsgOpt.Clear_P_Reset=TRUE
;Clear message on block selection
MsgOpt.Clear_p_SAW=FALSE
;Log message
MsgOpt.Log_To_DB=bLog

;set MessagNumber
Msg.Nr=nMsgNr
;set Msgtext
len=Strlen(sText[])
if len>0 then
	if len>80 then
		len=80
	endif
	for count=1 to len
		Msg.Msg_txt[count]=sText[count]
	endfor
else
	Msg.Msg_txt[]="Message text is missing"
endif
;setMsg-Modul
len=Strlen(sModul[])
if len>0 then
	if len>24 then
		len=24
	endif
	for count=1 to len
		Msg.Modul[count]=sModul[count]
	endfor
else
	Msg.Modul[]="Module name missing"
endif

CONTINUE
nHandle=Set_KrlMsg (MsgType, Msg, MsgPar[], MsgOpt)

END
;
;ENDFOLD (ISRA)

--- vw_isr_usr_r.dat ---
&ACCESS  RV
&COMMENT KS26
&PARAM DISKPATH = VW_User/Applikation/LM_Vision/Isra
&PARAM TPUSER_VERSION = 8.3.0
&PARAM EDITMASK = vw_isr_usr_r
&REL 59
DEFDAT  vw_isr_usr_r PUBLIC
;
;***************************************************
;* ISRA                                            *
;* Version 1.30  / VKRC 4                          *
;* Bearbeitet am:                                  *
;* 27.11.2014 JHo                                  *
;***************************************************
;
;FOLD IN-Signals IMT
; ;BYTE 0-3 / 4-7
SIGNAL IS_RX32_CORR_X $IN[1953]  TO $IN[1984] ;DATA-ID 52
SIGNAL IS_RX32_CORR_Y $IN[1985]  TO $IN[2016] ;DATA-ID 52
SIGNAL IS_RX32_CORR_Z $IN[1953]  TO $IN[1984] ;DATA-ID 53
SIGNAL IS_RX32_CORR_A $IN[1985]  TO $IN[2016] ;DATA-ID 53
SIGNAL IS_RX32_CORR_B $IN[1953]  TO $IN[1984] ;DATA-ID 54
SIGNAL IS_RX32_CORR_C $IN[1985]  TO $IN[2016] ;DATA-ID 54
;
SIGNAL IS_RX32_TOOL_X $IN[1953]  TO $IN[1984] ;DATA-ID 55
SIGNAL IS_RX32_TOOL_Y $IN[1985]  TO $IN[2016] ;DATA-ID 55
SIGNAL IS_RX32_TOOL_Z $IN[1953]  TO $IN[1984] ;DATA-ID 56
SIGNAL IS_RX32_TOOL_A $IN[1985]  TO $IN[2016] ;DATA-ID 56
SIGNAL IS_RX32_TOOL_B $IN[1953]  TO $IN[1984] ;DATA-ID 57
SIGNAL IS_RX32_TOOL_C $IN[1985]  TO $IN[2016] ;DATA-ID 57
;
;Error
SIGNAL IS_RX8_ERR_SYS_ID $IN[1953]  TO $IN[1960] ;DATA-ID 9/58
SIGNAL IS_RX8_ERRORS $IN[1961]  TO $IN[1968] ;DATA-ID 9/58
;
;State/Warnings
SIGNAL IS_RX8_STATE_RESULT $IN[1969]  TO $IN[1976] ;DATA-ID 58
SIGNAL IS_RX8_STATE_WARNING $IN[1977]  TO $IN[1984] ;DATA-ID 58
;
;BYTE 8
SIGNAL IS_RX8_DATA_ID $IN[2017]  TO $IN[2024]
;
;BYTE 9
SIGNAL IS_RX8_PROG_ID $IN[2025]  TO $IN[2032] ;Data-ID 51
;
;BYTE 10
SIGNAL IS_RX1_INIT_SIGNALS $IN[2033]
SIGNAL IS_RX1_SKIP $IN[2034]
SIGNAL IS_RX1_CONTINUE $IN[2035]
SIGNAL IS_RX1_MEAS_END $IN[2036] ;RF Messung Ende
;
;BYTE 11
SIGNAL IS_RX1_DATA_UNCHANGED $IN[2041]
SIGNAL IS_RX1_DATA_REQUEST $IN[2042]
SIGNAL IS_RX1_DATA_VALID $IN[2043]
SIGNAL IS_RX1_DATA_ACCEPTED $IN[2044]
SIGNAL IS_RX1_DATA_END_TRANS $IN[2045]
SIGNAL IS_RX1_ERROR_STATE $IN[2046]
SIGNAL IS_RX1_LIVE_SIGNAL $IN[2047]
SIGNAL IS_RX1_HANDSHAKE $IN[2048]
;
;ENDFOLD
;
;FOLD OUT-Signals IMT
;
;BYTE 0-3 / 4-7
SIGNAL IS_TX32_AXIS_1 $OUT[1953]  TO $OUT[1984] ;DATA-ID 1
SIGNAL IS_TX32_AXIS_2 $OUT[1985]  TO $OUT[2016] ;DATA-ID 1
SIGNAL IS_TX32_AXIS_3 $OUT[1953]  TO $OUT[1984] ;DATA-ID 2
SIGNAL IS_TX32_AXIS_4 $OUT[1985]  TO $OUT[2016] ;DATA-ID 2
SIGNAL IS_TX32_AXIS_5 $OUT[1953]  TO $OUT[1984] ;DATA-ID 3
SIGNAL IS_TX32_AXIS_6 $OUT[1985]  TO $OUT[2016] ;DATA-ID 3
;
SIGNAL IS_TX32_BASE_X $OUT[1953]  TO $OUT[1984] ;DATA-ID 4
SIGNAL IS_TX32_BASE_Y $OUT[1985]  TO $OUT[2016] ;DATA-ID 4
SIGNAL IS_TX32_BASE_Z $OUT[1953]  TO $OUT[1984] ;DATA-ID 5
SIGNAL IS_TX32_BASE_A $OUT[1985]  TO $OUT[2016] ;DATA-ID 5
SIGNAL IS_TX32_BASE_B $OUT[1953]  TO $OUT[1984] ;DATA-ID 6
SIGNAL IS_TX32_BASE_C $OUT[1985]  TO $OUT[2016] ;DATA-ID 6
;
SIGNAL IS_TX3_IMT_STATUS $OUT[1953]  TO $OUT[1960] ;DATA-ID 7
SIGNAL IS_TX6_IMT_TURN $OUT[1961]  TO $OUT[1968] ;DATA-ID 7
;
SIGNAL IS_TX8_MODEL_ID $OUT[1953]  TO $OUT[1960] ;DATA-ID 8
SIGNAL IS_TX8_ERROR_ID1 $OUT[1953]  TO $OUT[1960] ;DATA-ID 9
SIGNAL IS_TX8_ERROR_ID2 $OUT[1961]  TO $OUT[1968] ;DATA-ID 9
SIGNAL IS_TX16_SERVICE_ID $OUT[1953]  TO $OUT[1968] ;DATA-ID 10
;
SIGNAL IS_TX32_POSE_X $OUT[1953]  TO $OUT[1984] ;DATA-ID 11
SIGNAL IS_TX32_POSE_Y $OUT[1985]  TO $OUT[2016] ;DATA-ID 11
SIGNAL IS_TX32_POSE_Z $OUT[1953]  TO $OUT[1984] ;DATA-ID 12
SIGNAL IS_TX32_POSE_A $OUT[1985]  TO $OUT[2016] ;DATA-ID 12
SIGNAL IS_TX32_POSE_B $OUT[1953]  TO $OUT[1984] ;DATA-ID 13
SIGNAL IS_TX32_POSE_C $OUT[1985]  TO $OUT[2016] ;DATA-ID 13
;
SIGNAL IS_TX32_TOOL_X $OUT[1953]  TO $OUT[1984] ;DATA-ID 14
SIGNAL IS_TX32_TOOL_Y $OUT[1985]  TO $OUT[2016] ;DATA-ID 14
SIGNAL IS_TX32_TOOL_Z $OUT[1953]  TO $OUT[1984] ;DATA-ID 15
SIGNAL IS_TX32_TOOL_A $OUT[1985]  TO $OUT[2016] ;DATA-ID 15
SIGNAL IS_TX32_TOOL_B $OUT[1953]  TO $OUT[1984] ;DATA-ID 16
SIGNAL IS_TX32_TOOL_C $OUT[1985]  TO $OUT[2016] ;DATA-ID 16
;
;BYTE 8
SIGNAL IS_TX8_DATA_ID $OUT[2017]  TO $OUT[2024]
;
;BYTE 9
SIGNAL IS_TX8_POSE_ID $OUT[2025]  TO $OUT[2032]
;
;BYTE 10
SIGNAL IS_TX1_INIT_SIGNALS $OUT[2033]
SIGNAL IS_TX1_SKIP $OUT[2034]
SIGNAL IS_TX1_APPROACH_POSE $OUT[2035]
SIGNAL IS_TX1_IN_POSE $OUT[2036]
SIGNAL IS_TX1_IN_ENDPOSE $OUT[2037]
SIGNAL IS_TX1_TIMEOUT $OUT[2038]
;
;BYTE 11
SIGNAL IS_TX1_DATA_UNCHANGED $OUT[2041]
SIGNAL IS_TX1_DATA_REQUEST $OUT[2042]
SIGNAL IS_TX1_DATA_VALID $OUT[2043]
SIGNAL IS_TX1_DATA_ACCEPTED $OUT[2044]
SIGNAL IS_TX1_DATA_END_TRANS $OUT[2045]
SIGNAL IS_TX1_ERROR_STATE $OUT[2046]
SIGNAL IS_TX1_LIVE_BIT $OUT[2047]
SIGNAL IS_TX1_HANDSHAKE $OUT[2048]
;
;ENDFOLD
;
;FOLD IN-Signals RF
;
SIGNAL IS_RX4_RF_RM $IN[1953]  TO $IN[1956]
SIGNAL IS_RX1_RF_PREP_OK $IN[1960]
SIGNAL IS_RX1_RF_IMG_ACQ $IN[1957]
SIGNAL IS_RX1_RF_MEAS_RUN $IN[1958]
SIGNAL IS_RX1_RF_RES_RUN $IN[1959]
SIGNAL IS_RX1_RF_READY $IN[1961]
SIGNAL IS_RX1_RF_LIVE $IN[1962]
;
;Errors:
SIGNAL IS_RX1_RF_ERR_DEADLY $IN[1969]
SIGNAL IS_RX1_RF_ERR_PREP $IN[1973]
SIGNAL IS_RX1_RF_ERR_FEAT $IN[1972]
SIGNAL IS_RX1_RF_ERR_TOL $IN[1976]
SIGNAL IS_RX8_RF_ERR_SUM $IN[1969]  TO $IN[1976]
;
;Warnings:
SIGNAL IS_RX1_RF_W_MAN $IN[1977]
SIGNAL IS_RX1_RF_W_TOL $IN[1978]
SIGNAL IS_RX1_RF_W_EVAL $IN[1979]
;
;Result Data:
SIGNAL IS_RX16_RF_RES_X $IN[1985]  TO $IN[2000]
SIGNAL IS_RX16_RF_RES_Y $IN[2001]  TO $IN[2016]
SIGNAL IS_RX16_RF_RES_Z $IN[2017]  TO $IN[2032]
SIGNAL IS_RX16_RF_RES_RX $IN[2033]  TO $IN[2048]
SIGNAL IS_RX16_RF_RES_RY $IN[2049]  TO $IN[2064]
SIGNAL IS_RX16_RF_RES_RZ $IN[2065]  TO $IN[2080]
;
;ENDFOLD
;
;FOLD OUT-Signals RF
;
SIGNAL IS_TX4_RF_RM $OUT[1953]  TO $OUT[1956]
SIGNAL IS_TX1_RF_TYP_STR $OUT[1960]
SIGNAL IS_TX1_RF_START $OUT[1957]
SIGNAL IS_TX1_RF_SRESET $OUT[1958]
SIGNAL IS_TX1_RF_ERESET $OUT[1959]
SIGNAL IS_TX8_RF_TYP $OUT[1961]  TO $OUT[1968]
SIGNAL IS_TX8_RF_SUB_TYP $OUT[1969]  TO $OUT[1976]
SIGNAL IS_TX8_RF_COLOR_ID $OUT[1977]  TO $OUT[1984]
SIGNAL IS_TX1_RF_LIVE $OUT[1985]
;
SIGNAL IS_TX16_TYPE_ID $OUT[1953]  TO $OUT[1968] ;DATA-ID 8	;RF
SIGNAL IS_TX16_SUBTYPE_ID $OUT[1969]  TO $OUT[1984] ;DATA-ID 8	;RF
SIGNAL IS_TX16_COLOR_ID $OUT[1985]  TO $OUT[2000] ;DATA-ID 8	;RF
;
;ENDFOLD
;
;FOLD Constants
;
ENUM ISWaitType IS_NONE,IS_VALID,IS_ACCEPTED,IS_CONTINUE,IS_REQUEST,IS_END,IS_ERROR_ID,IS_RF_READY,IS_RF_RM,IS_RF_PREP,IS_RF_IMGACQ,IS_RF_MESRUN,IS_RF_ERESET,IS_RF_RESRUN
;
DECL REAL IS_RF_rScaleXYZ=10.0
DECL REAL IS_RF_rScaleABC=1000.0
DECL REAL IS_IMT_rScaleXYZ=100000.0
DECL REAL IS_IMT_rScaleABC=1000000.0
DECL REAL IS_IMT_rScaleAxis=1000000.0
DECL REAL IS_rSettlingTime=0.25 ; 250ms
;
DECL INT IS_iWaitTimerID=11
;
DECL INT IS_IMT_iRobStopTimerID=8
DECL INT IS_IMT_iRobStopTime=0
;
FRAME IS_CORR_ACCEPT_FRAME={X 20.0,Y 20.0,Z 20.0,A 5.0,B 5.0,C 5.0}
;
FRAME IS_ITERATION_THRESHOLD={X 0.0200000107,Y 0.0200000107,Z 0.0200000107,A 0.100000001,B 0.100000001,C 0.100000001}
;
;ENDFOLD
;
;FOLD Runtime Variables
;
DECL INT IS_ANSWER=2
CHAR IS_MG=" "
INT IS_MSG_I_LVL=0 ; 0-2 Message Level, um so hoeher das level, desto mehr meldungen.
;
DECL INT IS_MODUS
DECL INT IS_TYP
DECL INT IS_SUBTYP
DECL INT IS_SPECIFIER
DECL INT IS_TOOLNR
DECL INT IS_WIEDERHOLUNG
DECL INT IS_MODEL
DECL INT IS_PROGID
;
DECL INT IS_RX16_DATA[6]
;
DECL CHAR IS_strFnctName[20]
DECL CHAR IS_strErrText[32]
DECL CHAR IS_strErrorSource[10]
DECL CHAR IS_chCurrentFeature[100]
;
DECL BOOL IS_bHandshake=TRUE
DECL BOOL IS_bSkipFlag=FALSE
DECL BOOL IS_bTimeoutFlag=FALSE
DECL BOOL IS_bInternError
DECL BOOL IS_bSendBase=FALSE
DECL BOOL IS_bRepeatUpSel=FALSE
DECL BOOL IS_bMeasurementOK=FALSE
DECL BOOL IS_bSendAxes=TRUE
; HW error detection:
DECL BOOL IS_bHWCheckMode=FALSE
DECL BOOL IS_FLAGS_SAVED[13]
;
DECL INT IS_iCurrentUserError
DECL INT IS_iCurrentModel=70
DECL INT IS_iCurrentSub=70
DECL INT $IS_iHandshakeCounter=1
DECL INT IS_iErrorSource
DECL INT IS_iExternErrors
DECL INT IS_iInternErrors
DECL INT IS_iFnctID
DECL INT IS_iExternWarns_RF ;Warnzustände von RoVis für RF
;
DECL INT IS_iMeasPoint
;
DECL INT IS_iRM_Calib=1
;
DECL INT IS_iQuitFlag
;
DECL INT IS_iMaxNumIterations=1
;
DECL REAL IS_rMeasurementDelay
;
;ENDFOLD
;
;FOLD IDs
;
;Flags
DECL INT IS_FLAG_RESULT_OK=495
DECL INT IS_FLAG_RESULT_NOK=496
DECL INT IS_FLAG_ERROR=497
DECL INT IS_FLAG_ERR_SPS=498
DECL INT IS_FLAG_ERR_ROBOT=499
DECL INT IS_FLAG_ERR_PREPARE=500
DECL INT IS_FLAG_ERR_ACQ=501
DECL INT IS_FLAG_ERR_FEATURE=502
DECL INT IS_FLAG_ERR_EVAL=503
DECL INT IS_FLAG_ERR_TOL=504
DECL INT IS_FLAG_WARN_TOL=505
DECL INT IS_FLAG_KAL1_HLP=506
DECL INT IS_FLAG_KAL2_HLP=507
;
;Msg Type ID
DECL INT IS_MSG_TYPE_NOTIFY=1
DECL INT IS_MSG_TYPE_DIALOG=2
DECL INT IS_MSG_TYPE_QUIT=3
DECL INT IS_MSG_TYPE_STATE=4
;
;Msg ID User Instruction
DECL INT IS_MSG_PREP_INSTR=4002
DECL INT IS_MSG_ACQ_INSTR=4003
DECL INT IS_MSG_FEAT_INSTR=4004
DECL INT IS_MSG_EVAL_INSTR=4005
DECL INT IS_MSG_TOL_INSTR=4006
;
;Msg ID Info
DECL INT IS_MSG_I_SERV_SENS_CHK=2003
DECL INT IS_MSG_I_SERV_SENS=2004
DECL INT IS_MSG_I_SERV_TOOL=2005
DECL INT IS_MSG_I_SERV_TOOL_PATH1=2006
DECL INT IS_MSG_I_SERV_ROB=2007
DECL INT IS_MSG_I_SERV_ROB_PATH1=2008
DECL INT IS_MSG_I_SERV_SENSIMT=2009
DECL INT IS_MSG_I_TRANS_AXES=2010
DECL INT IS_MSG_I_TRANS_BASE=2011
DECL INT IS_MSG_I_SYS_DIAG_1=3000
DECL INT IS_MSG_I_SYS_DIAG_2=3001
DECL INT IS_MSG_I_SYS_DIAG_3=3002
DECL INT IS_MSG_I_SYS_DIAG_4=3003
DECL INT IS_MSG_I_SYS_DIAG_5=3004
DECL INT IS_MSG_I_SYS_DIAG_6=3005
DECL INT IS_MSG_I_SYS_DIAG_7=3006
DECL INT IS_MSG_I_SYNC=4001 ; 7
DECL INT IS_MSG_I_MEAS_FAILED=4002 ; 8
DECL INT IS_MSG_I_SERV_TOOL_PATH2=4003 ; 12
DECL INT IS_MSG_I_SERV_ROB_PATH2=4004 ; 13
;
;Msg ID Error
DECL INT IS_MSG_ERR_SYNC1A=200
DECL INT IS_MSG_ERR_SYNC1B=201
DECL INT IS_MSG_ERR_SYNC2A=202
DECL INT IS_MSG_ERR_SYNC2B=203
DECL INT IS_MSG_ERR_SELECT1=204
DECL INT IS_MSG_ERR_SELECT1A=205
DECL INT IS_MSG_ERR_SELECT1B=206
DECL INT IS_MSG_ERR_SELECT1C=207
DECL INT IS_MSG_ERR_SELECT2=208
DECL INT IS_MSG_ERR_SELECT2A=209
DECL INT IS_MSG_ERR_SELECT2B=210
DECL INT IS_MSG_ERR_SELECT3=211
DECL INT IS_MSG_ERR_SELECT3A=212
DECL INT IS_MSG_ERR_IMT_PREPARE1=213
DECL INT IS_MSG_ERR_IMT_PREPARE1A=214
DECL INT IS_MSG_ERR_IMT_PREPARE1B=215
DECL INT IS_MSG_ERR_IMT_APPLY=216
DECL INT IS_MSG_ERR_AXIS1=217
DECL INT IS_MSG_ERR_AXIS1A=218
DECL INT IS_MSG_ERR_AXIS1B=219
DECL INT IS_MSG_ERR_AXIS1C=220
DECL INT IS_MSG_ERR_AXIS1D=221
DECL INT IS_MSG_ERR_AXIS2=222
DECL INT IS_MSG_ERR_AXIS2A=223
DECL INT IS_MSG_ERR_AXIS2B=224
DECL INT IS_MSG_ERR_AXIS3=225
DECL INT IS_MSG_ERR_AXIS3A=226
DECL INT IS_MSG_ERR_AXIS3B=227
DECL INT IS_MSG_ERR_AXIS4=228
DECL INT IS_MSG_ERR_AXIS4A=229
DECL INT IS_MSG_ERR_AXIS4B=230
DECL INT IS_MSG_ERR_BASE1=231
DECL INT IS_MSG_ERR_BASE1A=232
DECL INT IS_MSG_ERR_BASE1B=233
DECL INT IS_MSG_ERR_BASE2=234
DECL INT IS_MSG_ERR_BASE2A=235
DECL INT IS_MSG_ERR_BASE2B=236
DECL INT IS_MSG_ERR_BASE3=237
DECL INT IS_MSG_ERR_BASE3A=238
DECL INT IS_MSG_ERR_BASE3B=239
DECL INT IS_MSG_ERR_IMT_END1=240
DECL INT IS_MSG_ERR_IMT_END1A=241
DECL INT IS_MSG_ERR_IMT_END1B=242
DECL INT IS_MSG_ERR_IMT_END1C=243
DECL INT IS_MSG_ERR_GETCORR1=244
DECL INT IS_MSG_ERR_GETCORR1A=245
DECL INT IS_MSG_ERR_GETCORR1B=246
DECL INT IS_MSG_ERR_GETCORR2=247
DECL INT IS_MSG_ERR_GETCORR2A=248
DECL INT IS_MSG_ERR_GETCORR2B=249
DECL INT IS_MSG_ERR_GETCORR3=250
DECL INT IS_MSG_ERR_GETCORR3A=251
DECL INT IS_MSG_ERR_GETCORR3B=252
DECL INT IS_MSG_ERR_GETCORR4=253
DECL INT IS_MSG_ERR_GETCORR4A=254
DECL INT IS_MSG_ERR_POSE1=255
DECL INT IS_MSG_ERR_POSE1A=256
DECL INT IS_MSG_ERR_POSE1B=257
DECL INT IS_MSG_ERR_POSE2=258
DECL INT IS_MSG_ERR_POSE2A=259
DECL INT IS_MSG_ERR_POSE2B=260
DECL INT IS_MSG_ERR_POSE3=261
DECL INT IS_MSG_ERR_POSE3A=262
DECL INT IS_MSG_ERR_POSE3B=263
DECL INT IS_MSG_ERR_TOOL1=264
DECL INT IS_MSG_ERR_TOOL1A=265
DECL INT IS_MSG_ERR_TOOL1B=266
DECL INT IS_MSG_ERR_TOOL2=267
DECL INT IS_MSG_ERR_TOOL2A=268
DECL INT IS_MSG_ERR_TOOL2B=269
DECL INT IS_MSG_ERR_TOOL3=270
DECL INT IS_MSG_ERR_TOOL3A=271
DECL INT IS_MSG_ERR_TOOL3B=272
;
DECL INT IS_MSG_ERR_RTC=277
DECL INT IS_MSG_ERR_RTC_CALIB=278
DECL INT IS_MSG_ERR_RTC_CALC_TOOL=279
DECL INT IS_MSG_ERR_RTC_CALC_BASE=280
DECL INT IS_MSG_ERR_SERV_SENS1=281
DECL INT IS_MSG_ERR_SERV_SENS2=282
DECL INT IS_MSG_ERR_SERV_TOOL=283
DECL INT IS_MSG_ERR_SERV_ROB=284
DECL INT IS_MSG_ERR_SERV_SENSIMT=285
DECL INT IS_MSG_ERR_SERV_ROB_C=286
DECL INT IS_MSG_ERR_SERV_TOOL_C=287
DECL INT IS_MSG_ERR_SERV_ROB_T=288
DECL INT IS_MSG_ERR_SERV_TOOL_T=289
;
DECL INT IS_MSG_ERR_TOL_EXCEEDED=291
;RF
DECL INT IS_MSG_ERR_RF_INIT1A=299
DECL INT IS_MSG_ERR_RF_INIT2A=300
DECL INT IS_MSG_ERR_RF_PREPARE1=301
DECL INT IS_MSG_ERR_RF_PREPARE1A=302
DECL INT IS_MSG_ERR_RF_PREPARE1B=303
DECL INT IS_MSG_ERR_RF_PREPARE2=304
DECL INT IS_MSG_ERR_RF_PREPARE2A=305
DECL INT IS_MSG_ERR_RF_PREPARE2B=306
DECL INT IS_MSG_ERR_RF_PREPARE3=307
DECL INT IS_MSG_ERR_RF_PREPARE3A=308
DECL INT IS_MSG_ERR_RF_PREPARE3B=309
DECL INT IS_MSG_ERR_RF_PREPARE3C=310
DECL INT IS_MSG_ERR_RF_APPLY1=311
DECL INT IS_MSG_ERR_RF_APPLY2=312
DECL INT IS_MSG_ERR_RF_APPLY2A=313
DECL INT IS_MSG_ERR_RF_APPLY2B=314
DECL INT IS_MSG_ERR_RF_APPLY3=315
DECL INT IS_MSG_ERR_RF_APPLY3A=316
DECL INT IS_MSG_ERR_RF_APPLY3B=317
DECL INT IS_MSG_ERR_RF_APPLY3C=318
DECL INT IS_MSG_ERR_RF_APPLY3D=319
DECL INT IS_MSG_ERR_RF_APPLY3E=320
DECL INT IS_MSG_ERR_RF_APPLY4=321
DECL INT IS_MSG_ERR_RF_APPLY4A=322
DECL INT IS_MSG_ERR_RF_APPLY4B=323
DECL INT IS_MSG_ERR_RF_APPLY4C=324
DECL INT IS_MSG_ERR_RF_APPLY4D=325
DECL INT IS_MSG_ERR_RF_APPLY4E=326
DECL INT IS_MSG_ERR_RF_APPLY5=327
DECL INT IS_MSG_ERR_RF_APPLY5A=328
DECL INT IS_MSG_ERR_RF_APPLY5B=329
DECL INT IS_MSG_ERR_RF_APPLY5C=330
DECL INT IS_MSG_ERR_RF_APPLY5D=331
DECL INT IS_MSG_ERR_RF_APPLY5E=332
DECL INT IS_MSG_ERR_RF_APPLY6=333
DECL INT IS_MSG_ERR_RF_END1=334
DECL INT IS_MSG_ERR_RF_END1A=335
DECL INT IS_MSG_ERR_RF_END1B=336
DECL INT IS_MSG_ERR_RF_END1C=337
DECL INT IS_MSG_ERR_RF_END1D=338
DECL INT IS_MSG_ERR_RF_END1E=339
DECL INT IS_MSG_ERR_RF_END2=340
DECL INT IS_MSG_ERR_RF_END2A=341
DECL INT IS_MSG_ERR_RF_END2B=342
DECL INT IS_MSG_ERR_RF_END2C=343
DECL INT IS_MSG_ERR_RF_END2D=344
DECL INT IS_MSG_ERR_RF_END2E=345
DECL INT IS_MSG_ERR_RF_END3=346
DECL INT IS_MSG_ERR_RF_CORR1=347
DECL INT IS_MSG_ERR_RF_CORR1A=348
DECL INT IS_MSG_ERR_RF_CORR1B=349
DECL INT IS_MSG_ERR_RF_CORR2=350
DECL INT IS_MSG_ERR_RF_CORR2A=351
DECL INT IS_MSG_ERR_RF_CORR2B=352
DECL INT IS_MSG_ERR_RF_CORR3=353
DECL INT IS_MSG_ERR_SERVICE1A=400
DECL INT IS_MSG_ERR_SERVICE1B=401
DECL INT IS_MSG_ERR_SERVICE1C=402
DECL INT IS_MSG_ERR_SERVICE1D=403
DECL INT IS_MSG_ERR_SERVICE1E=404
DECL INT IS_MSG_ERR_SERVICE1F=405
DECL INT IS_MSG_ERR_SERVICE1G=406
DECL INT IS_MSG_ERR_SERVICE1H=407
;
DECL INT IS_MSG_RESULT_OK=500
DECL INT IS_MSG_RESULT_NOK=501
DECL INT IS_MSG_WARN_TOL=502
;
; NEU fuer IMT
DECL INT IS_MSG_ERR_REQUEST=613
DECL INT IS_MSG_ERR_BASE=617
DECL INT IS_MSG_ERR_BIT_TRNS=619
DECL INT IS_MSG_ERR_TRANSM=629
DECL INT IS_MSG_PP_WARN=630
DECL INT IS_MSG_PP_MOVEMODE=361
DECL INT IS_MSG_PP_TOL=632
DECL INT IS_MSG_PP_INVERSE=633
DECL INT IS_MSG_PP_FORWARD=634
DECL INT IS_MSG_PP_TEST_POSA=635
DECL INT IS_MSG_PP_TEST_POSK=636
DECL INT IS_MSG_WAIT_LOOP1=637
DECL INT IS_MSG_WAIT_LOOP2=638
;
DECL INT IS_MSG_DEBUG=1500
DECL INT IS_MSG_ERR_DEFAULT=1501
;
;ID's for user instruction
DECL INT IS_Instr_Response=1 ;Das ISRA-System antwortet nicht. Prüfen Sie den Zustand des ISRA-Systems
DECL INT IS_Instr_ModelCmp=2 ;Vergleichen Sie die Modellnummern zwischen dem ISRA-System und dem Roboter
DECL INT IS_Instr_ModelChk=3 ;Prüfen Sie im ISRA-System, ob das Modell vorhanden und aktiviert ist
DECL INT IS_Instr_DeadlyErr=4 ;Schwerwiegender Ablauffehler: Bitte führen Sie einen Neustart oder eine Reinitialisierung des ISRA-Systems aus
DECL INT IS_Instr_RoutCheck=5 ;Vergleichen Sie die RoutinenNr zwischen dem ISRA-System und dem Roboter
DECL INT IS_Instr_PntChk=6 ;Legen Sie den Messpunkt im ISRA-System an, oder prüfen Sie die ID's
DECL INT IS_Instr_TolChk=7 ;Prüfen Sie die eingestellten Grenzen im ISRA-System
DECL INT IS_Instr_CalChk=8 ;Prüfen Sie das letzte Ergebnis der Kalibrierung in DynaFlexI
DECL INT IS_Instr_ImgMsgChk=9 ;Überprüfen Sie das Messbild sowie die Ausgaben im ISRA-System
DECL INT IS_Instr_RobTol=10 ;Passen Sie ggf. die Toleranz über die Variable IS_CORR_ACCEPT_FRAME an
DECL INT IS_Instr_TypeChk=11 ;Prüfen Sie im ISRA-System, ob der Typ vorhanden und aktiviert ist
DECL INT IS_Instr_HWChk=12 ;Prüfen Sie den Anschluss der Kamera(s)
DECL INT IS_Instr_MsgChk=13 ;Prüfen Sie die Ausgaben des ISRA-Systems
DECL INT IS_Instr_RobProg=14 ;Prüfen Sie die Messaufrufe im Roboterprogramm
;
;Error IDs VW-User
DECL INT IS_Err_ID=1 ;NOT USED
DECL INT IS_Err_ID_Com=2 ;NOT USED
DECL INT IS_Err_ID_Drain=3
DECL INT IS_Err_ID_Timeout=4
DECL INT IS_Err_ID_ProgID=5
DECL INT IS_Err_ID_Tolerance=6
;
; ISRA Intern Errors
DECL INT IS_IntErr_Param1=1000
DECL INT IS_IntErr_Param2=1001
DECL INT IS_IntErr_Param3=1002
DECL INT IS_IntErr_Param4=1003
DECL INT IS_IntErr_Param5=1004
DECL INT IS_IntErr_Param6=1005
DECL INT IS_IntErr_Com=1010
DECL INT IS_IntErr_ERequest=1013
DECL INT IS_IntErr_Meas=1014 ;NOT USED
DECL INT IS_IntErr_Retry=1015 ;NOT USED
DECL INT IS_IntErr_Data=1016 ;NOT USED
DECL INT IS_IntErr_Base=1017
DECL INT IS_IntErr_Tool=1018
DECL INT IS_IntErr_ESendBit=1019
DECL INT IS_IntErr_Specif=1020
DECL INT IS_IntErr_SrvcExp=1021
DECL INT IS_IntErr_StReq1=1023
DECL INT IS_IntErr_StReq2=1024
DECL INT IS_IntErr_ESend=1026
DECL INT IS_IntErr_IQRWait=1030 ;NOT USED
DECL INT IS_IntErr_PCWait=1031 ;NOT USED
DECL INT IS_IntErr_TolRob=1032
DECL INT IS_IntErr_RFAState=1033
DECL INT IS_IntErr_MeasPosNo=1034
DECL INT IS_IntErr_RFGCSt=1035
DECL INT IS_IntErr_RFEPSt=1036
;
;ISRA Error Bits (ROVIS internal - nur f?r RF relevant)
DECL INT IS_ErrBit_SPS=1
DECL INT IS_ErrBit_Rob=2
DECL INT IS_ErrBit_Command=4
DECL INT IS_ErrBit_Deadly=4 ; TODO
DECL INT IS_ErrBit_Prepare=8
DECL INT IS_ErrBit_ACQ=16
DECL INT IS_ErrBit_Axis=16 ; not RoVis
DECL INT IS_ErrBit_Feature=32
DECL INT IS_ErrBit_Base=32 ; not RoVis
DECL INT IS_ErrBit_Eval=64
DECL INT IS_ErrBit_Tol=128
;
;ISRA State IDs
DECL INT IS_STATE_RESULT_OK=1 ; not RoVis
DECL INT IS_STATE_RESULT_NOK=2 ; not RoVis
DECL INT IS_STATE_WARN_MANMEAS=1
DECL INT IS_STATE_WARN_RELIABLTY=2
DECL INT IS_STATE_WARN_EVAL=4
DECL INT IS_STATE_WARN_TOL=8
DECL INT IS_STATE_WARN_SENSOR=16
DECL INT IS_STATE_WARN_FEATURE=32
;
;FunctionIDs (nach Vorlage FANUC)
DECL INT IS_FnctID_IMT_Sync1=1
DECL INT IS_FnctID_IMT_Sync2=2
DECL INT IS_FnctID_IMT_SelectUp1=3
DECL INT IS_FnctID_IMT_SelectUp2=4
DECL INT IS_FnctID_IMT_SelectUp3=5
DECL INT IS_FnctID_IMT_GetCorr1=6
DECL INT IS_FnctID_IMT_GetCorr2=7
DECL INT IS_FnctID_IMT_GetCorr3=8
DECL INT IS_FnctID_IMT_GetCorr4=9
DECL INT IS_FnctID_IMT_Prepare=13
DECL INT IS_FnctID_IMT_Apply=14
DECL INT IS_FnctID_IMT_SendAxis1=15
DECL INT IS_FnctID_IMT_SendAxis2=16
DECL INT IS_FnctID_IMT_SendAxis3=17
DECL INT IS_FnctID_IMT_SendAxis4=18
DECL INT IS_FnctID_IMT_SendBase1=19
DECL INT IS_FnctID_IMT_SendBase2=20
DECL INT IS_FnctID_IMT_SendBase3=21
DECL INT IS_FnctID_IMT_EndPose1=22
DECL INT IS_FnctID_IMT_EndPose2=23
DECL INT IS_FnctID_IMT_SetError=24 ; NOT USED
DECL INT IS_FnctID_IMT_GetExtErr=25
DECL INT IS_FnctID_IMT_GetExtStat=26
DECL INT IS_FnctID_IMT_SendPose1=27
DECL INT IS_FnctID_IMT_SendPose2=28
DECL INT IS_FnctID_IMT_SendPose3=29
DECL INT IS_FnctID_IMT_SendTool1=30
DECL INT IS_FnctID_IMT_SendTool2=31
DECL INT IS_FnctID_IMT_SendTool3=32
DECL INT IS_FnctID_IMT_Service=33 ;27
DECL INT IS_FnctID_RF_End1=34 ;28
DECL INT IS_FnctID_RF_End2=35 ;29
DECL INT IS_FnctID_RF_End3=36 ;30
DECL INT IS_FnctID_RF_Prepare1=37 ;31
DECL INT IS_FnctID_RF_Prepare2=38 ;32
DECL INT IS_FnctID_RF_Prepare3=39 ;33
DECL INT IS_FnctID_RF_Apply1=40
DECL INT IS_FnctID_RF_Apply2=41
DECL INT IS_FnctID_RF_Apply3=42
DECL INT IS_FnctID_RF_Apply4=43
DECL INT IS_FnctID_RF_Apply5=44
DECL INT IS_FnctID_RF_Apply6=45
DECL INT IS_FnctID_RF_Init1=50
DECL INT IS_FnctID_RF_Init2=51
DECL INT IS_FnctID_RF_GCorr1=60
DECL INT IS_FnctID_RF_GCorr2=61
DECL INT IS_FnctID_RF_GCorr3=62
;
;ENDFOLD
;
;Fold UP-Nummerzuweisung 				---TODO
DECL INT UPNR[100,50] ; [Modellnr, Routinennr]
;Modell 10
UPNR[10,10]=10
UPNR[10,11]=11
UPNR[10,12]=12
UPNR[10,13]=13
UPNR[10,14]=14
UPNR[10,15]=15
UPNR[10,16]=16
UPNR[10,30]=80
UPNR[10,31]=81
UPNR[10,32]=82
UPNR[10,33]=83
UPNR[10,34]=84
UPNR[10,35]=85
UPNR[10,36]=86
UPNR[10,37]=87
UPNR[10,38]=88
UPNR[10,39]=89
UPNR[10,40]=90
UPNR[10,41]=91
UPNR[10,42]=92
UPNR[10,43]=93
UPNR[10,44]=94
;Kalib
UPNR[100,30]=80
UPNR[100,31]=81
UPNR[100,32]=82
UPNR[100,33]=83
UPNR[100,34]=84
UPNR[100,35]=85
UPNR[100,36]=86
UPNR[100,37]=87
UPNR[100,38]=88
UPNR[100,39]=89
UPNR[100,40]=90
UPNR[100,41]=91
UPNR[100,42]=92
UPNR[100,43]=93
UPNR[100,44]=94
;
;ENDFOLD
;
ENDDAT
